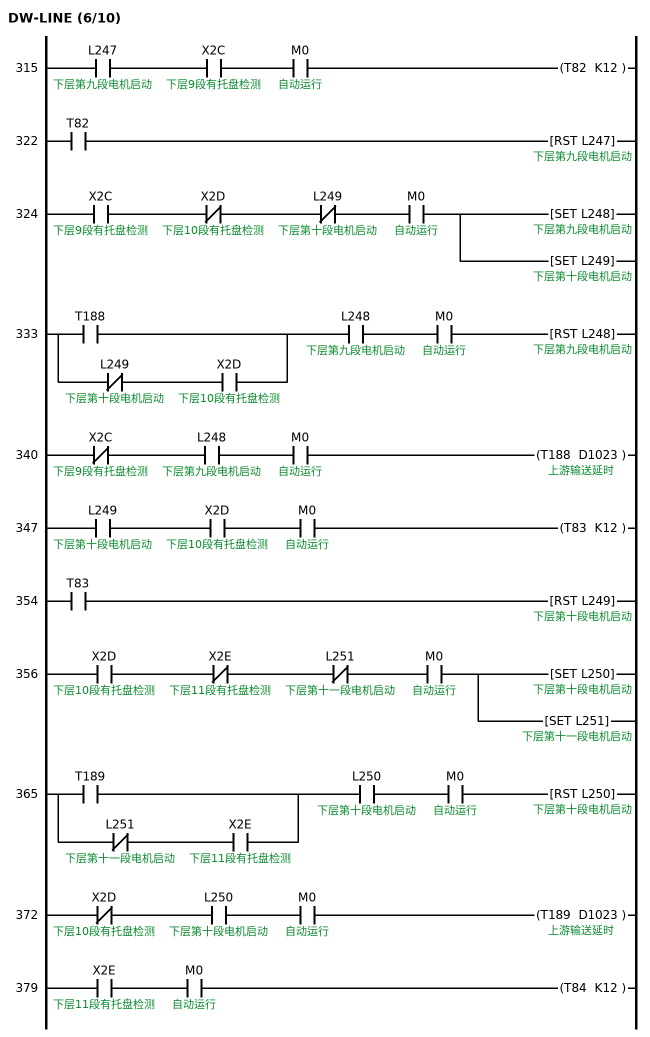
[picture p24: ladder of DW-LINE, rungs at steps 315 to 379]
315   LD      L247  ; 下层第九段电机启动
      AND     X2C  ; 下层9段有托盘检测
      AND     M0  ; 自动运行
      OUT     T82 K12
322   LD      T82
      RST     L247  ; 下层第九段电机启动
324   LD      X2C  ; 下层9段有托盘检测
      ANI     X2D  ; 下层10段有托盘检测
      ANI     L249  ; 下层第十段电机启动
      AND     M0  ; 自动运行
      SET     L248  ; 下层第九段电机启动
        [note] 10
      SET     L249  ; 下层第十段电机启动
333   LD      T188
      LDI     L249  ; 下层第十段电机启动
      AND     X2D  ; 下层10段有托盘检测
      ORB
      AND     L248  ; 下层第九段电机启动
      AND     M0  ; 自动运行
      RST     L248  ; 下层第九段电机启动
340   LDI     X2C  ; 下层9段有托盘检测
      AND     L248  ; 下层第九段电机启动
      AND     M0  ; 自动运行
      OUT     T188 D1023  ; 上游输送延时
347   LD      L249  ; 下层第十段电机启动
      AND     X2D  ; 下层10段有托盘检测
      AND     M0  ; 自动运行
      OUT     T83 K12
354   LD      T83
      RST     L249  ; 下层第十段电机启动
356   LD      X2D  ; 下层10段有托盘检测
      ANI     X2E  ; 下层11段有托盘检测
      ANI     L251  ; 下层第十一段电机启动
      AND     M0  ; 自动运行
      SET     L250  ; 下层第十段电机启动
        [note] 10
      SET     L251  ; 下层第十一段电机启动
365   LD      T189
      LDI     L251  ; 下层第十一段电机启动
      AND     X2E  ; 下层11段有托盘检测
      ORB
      AND     L250  ; 下层第十段电机启动
      AND     M0  ; 自动运行
      RST     L250  ; 下层第十段电机启动
372   LDI     X2D  ; 下层10段有托盘检测
      AND     L250  ; 下层第十段电机启动
      AND     M0  ; 自动运行
      OUT     T189 D1023  ; 上游输送延时
379   LD      X2E  ; 下层11段有托盘检测
      AND     M0  ; 自动运行
      OUT     T84 K12
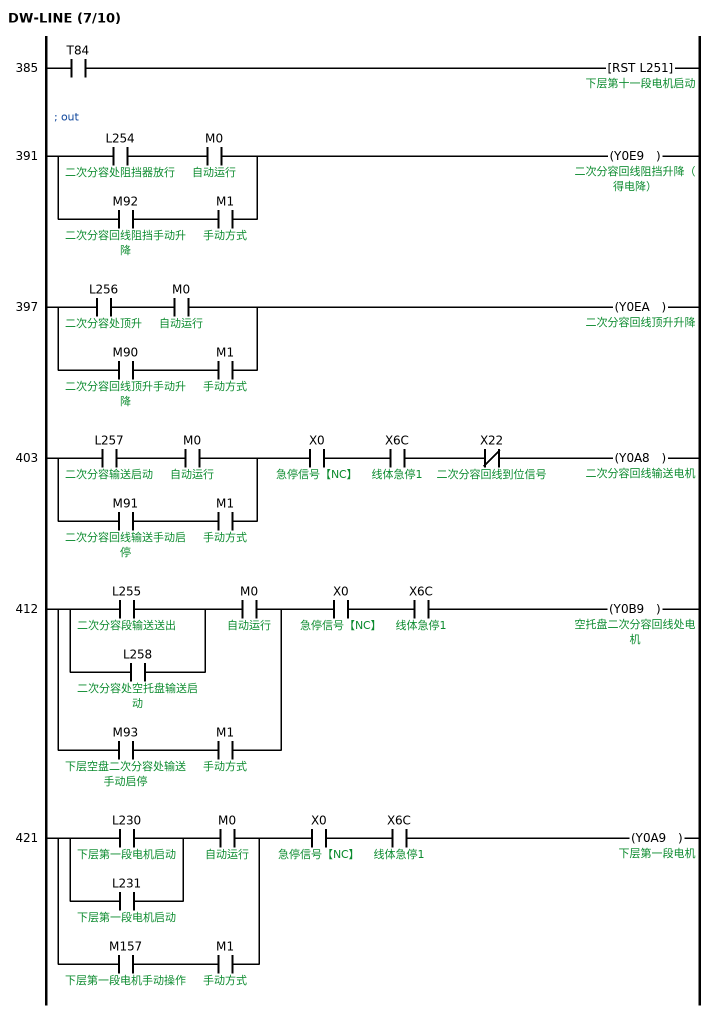
385   LD      T84
      RST     L251  ; 下层第十一段电机启动
; out
391   LD      L254  ; 二次分容处阻挡器放行
      AND     M0  ; 自动运行
      LD      M92  ; 二次分容回线阻挡手动升降
      AND     M1  ; 手动方式
      ORB
      OUT     Y0E9  ; 二次分容回线阻挡升降（得电降）
397   LD      L256  ; 二次分容处顶升
      AND     M0  ; 自动运行
      LD      M90  ; 二次分容回线顶升手动升降
      AND     M1  ; 手动方式
      ORB
      OUT     Y0EA  ; 二次分容回线顶升升降
403   LD      L257  ; 二次分容输送启动
      AND     M0  ; 自动运行
      LD      M91  ; 二次分容回线输送手动启停
      AND     M1  ; 手动方式
      ORB
      AND     X0  ; 急停信号【NC】
      AND     X6C  ; 线体急停1
      ANI     X22  ; 二次分容回线到位信号
      OUT     Y0A8  ; 二次分容回线输送电机
412   LD      L255  ; 二次分容段输送送出
      OR      L258  ; 二次分容处空托盘输送启动
      AND     M0  ; 自动运行
      LD      M93  ; 下层空盘二次分容处输送手动启停
      AND     M1  ; 手动方式
      ORB
      AND     X0  ; 急停信号【NC】
      AND     X6C  ; 线体急停1
      OUT     Y0B9  ; 空托盘二次分容回线处电机
421   LD      L230  ; 下层第一段电机启动
      OR      L231  ; 下层第一段电机启动
      AND     M0  ; 自动运行
      LD      M157  ; 下层第一段电机手动操作
      AND     M1  ; 手动方式
      ORB
      AND     X0  ; 急停信号【NC】
      AND     X6C  ; 线体急停1
      OUT     Y0A9  ; 下层第一段电机
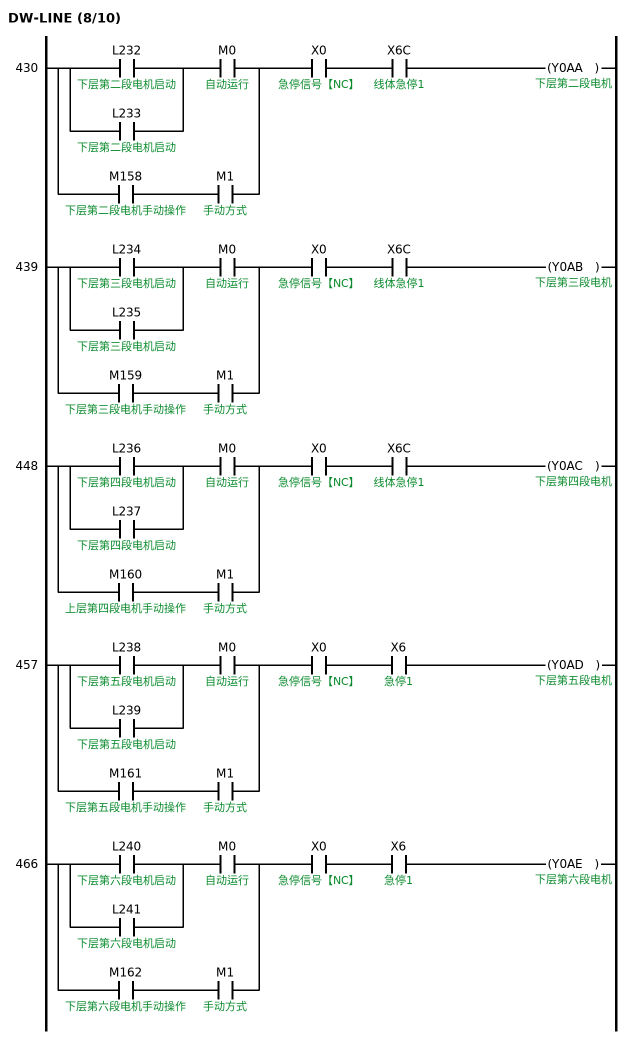
430   LD      L232  ; 下层第二段电机启动
      OR      L233  ; 下层第二段电机启动
      AND     M0  ; 自动运行
      LD      M158  ; 下层第二段电机手动操作
      AND     M1  ; 手动方式
      ORB
      AND     X0  ; 急停信号【NC】
      AND     X6C  ; 线体急停1
      OUT     Y0AA  ; 下层第二段电机
439   LD      L234  ; 下层第三段电机启动
      OR      L235  ; 下层第三段电机启动
      AND     M0  ; 自动运行
      LD      M159  ; 下层第三段电机手动操作
      AND     M1  ; 手动方式
      ORB
      AND     X0  ; 急停信号【NC】
      AND     X6C  ; 线体急停1
      OUT     Y0AB  ; 下层第三段电机
448   LD      L236  ; 下层第四段电机启动
      OR      L237  ; 下层第四段电机启动
      AND     M0  ; 自动运行
      LD      M160  ; 上层第四段电机手动操作
      AND     M1  ; 手动方式
      ORB
      AND     X0  ; 急停信号【NC】
      AND     X6C  ; 线体急停1
      OUT     Y0AC  ; 下层第四段电机
457   LD      L238  ; 下层第五段电机启动
      OR      L239  ; 下层第五段电机启动
      AND     M0  ; 自动运行
      LD      M161  ; 下层第五段电机手动操作
      AND     M1  ; 手动方式
      ORB
      AND     X0  ; 急停信号【NC】
      AND     X6  ; 急停1
      OUT     Y0AD  ; 下层第五段电机
466   LD      L240  ; 下层第六段电机启动
      OR      L241  ; 下层第六段电机启动
      AND     M0  ; 自动运行
      LD      M162  ; 下层第六段电机手动操作
      AND     M1  ; 手动方式
      ORB
      AND     X0  ; 急停信号【NC】
      AND     X6  ; 急停1
      OUT     Y0AE  ; 下层第六段电机
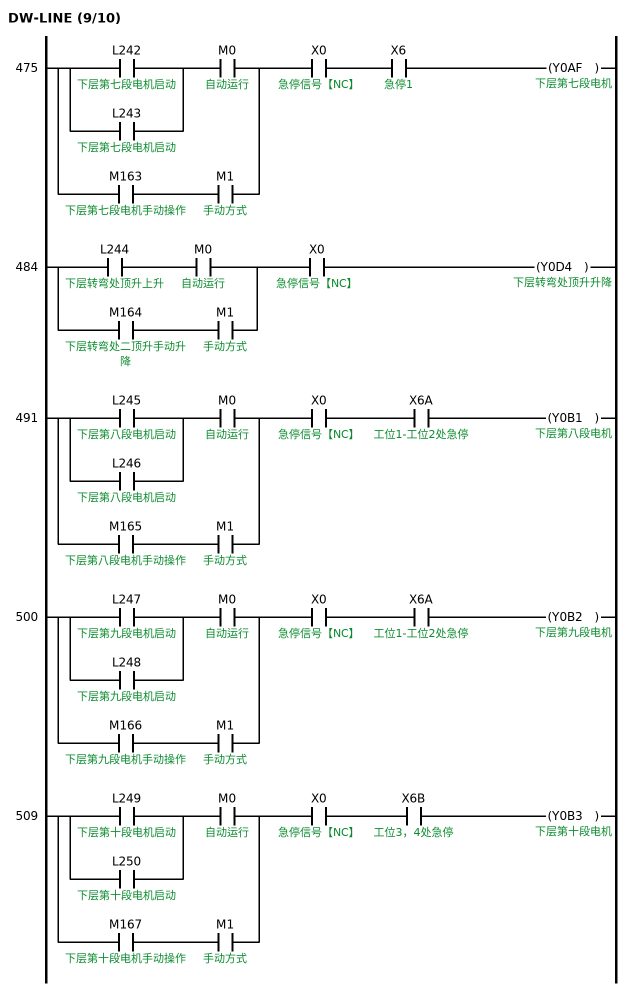
475   LD      L242  ; 下层第七段电机启动
      OR      L243  ; 下层第七段电机启动
      AND     M0  ; 自动运行
      LD      M163  ; 下层第七段电机手动操作
      AND     M1  ; 手动方式
      ORB
      AND     X0  ; 急停信号【NC】
      AND     X6  ; 急停1
      OUT     Y0AF  ; 下层第七段电机
484   LD      L244  ; 下层转弯处顶升上升
      AND     M0  ; 自动运行
      LD      M164  ; 下层转弯处二顶升手动升降
      AND     M1  ; 手动方式
      ORB
      AND     X0  ; 急停信号【NC】
      OUT     Y0D4  ; 下层转弯处顶升升降
491   LD      L245  ; 下层第八段电机启动
      OR      L246  ; 下层第八段电机启动
      AND     M0  ; 自动运行
      LD      M165  ; 下层第八段电机手动操作
      AND     M1  ; 手动方式
      ORB
      AND     X0  ; 急停信号【NC】
      AND     X6A  ; 工位1-工位2处急停
      OUT     Y0B1  ; 下层第八段电机
500   LD      L247  ; 下层第九段电机启动
      OR      L248  ; 下层第九段电机启动
      AND     M0  ; 自动运行
      LD      M166  ; 下层第九段电机手动操作
      AND     M1  ; 手动方式
      ORB
      AND     X0  ; 急停信号【NC】
      AND     X6A  ; 工位1-工位2处急停
      OUT     Y0B2  ; 下层第九段电机
509   LD      L249  ; 下层第十段电机启动
      OR      L250  ; 下层第十段电机启动
      AND     M0  ; 自动运行
      LD      M167  ; 下层第十段电机手动操作
      AND     M1  ; 手动方式
      ORB
      AND     X0  ; 急停信号【NC】
      AND     X6B  ; 工位3，4处急停
      OUT     Y0B3  ; 下层第十段电机
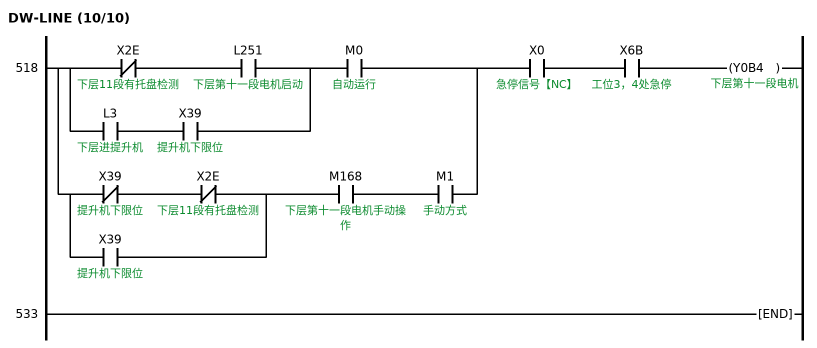
518   LDI     X2E  ; 下层11段有托盘检测
      AND     L251  ; 下层第十一段电机启动
      LD      L3  ; 下层进提升机
      AND     X39  ; 提升机下限位
      ORB
      AND     M0  ; 自动运行
      LDI     X39  ; 提升机下限位
      ANI     X2E  ; 下层11段有托盘检测
      OR      X39  ; 提升机下限位
      AND     M168  ; 下层第十一段电机手动操作
      AND     M1  ; 手动方式
      ORB
      AND     X0  ; 急停信号【NC】
      AND     X6B  ; 工位3，4处急停
      OUT     Y0B4  ; 下层第十一段电机
533   END
END_PROGRAM

PROGRAM ELEVATR
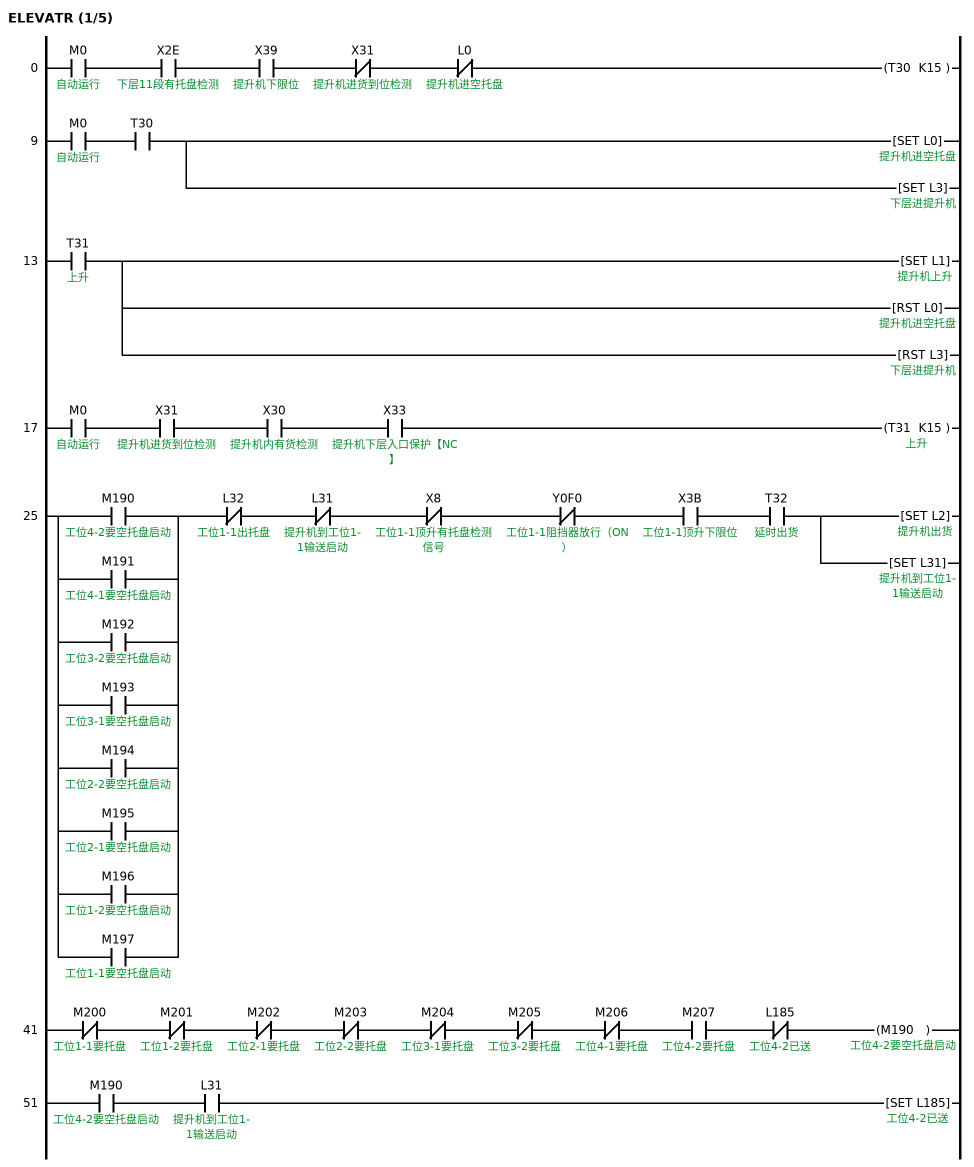
0     LD      M0  ; 自动运行
      AND     X2E  ; 下层11段有托盘检测
      AND     X39  ; 提升机下限位
      ANI     X31  ; 提升机进货到位检测
      ANI     L0  ; 提升机进空托盘
      OUT     T30 K15
9     LD      M0  ; 自动运行
      AND     T30
      SET     L0  ; 提升机进空托盘
      SET     L3  ; 下层进提升机
13    LD      T31  ; 上升
      SET     L1  ; 提升机上升
      RST     L0  ; 提升机进空托盘
      RST     L3  ; 下层进提升机
17    LD      M0  ; 自动运行
      AND     X31  ; 提升机进货到位检测
      AND     X30  ; 提升机内有货检测
      AND     X33  ; 提升机下层入口保护【NC】
      OUT     T31 K15  ; 上升
25    LD      M190  ; 工位4-2要空托盘启动
      OR      M191  ; 工位4-1要空托盘启动
      OR      M192  ; 工位3-2要空托盘启动
      OR      M193  ; 工位3-1要空托盘启动
      OR      M194  ; 工位2-2要空托盘启动
      OR      M195  ; 工位2-1要空托盘启动
      OR      M196  ; 工位1-2要空托盘启动
      OR      M197  ; 工位1-1要空托盘启动
      ANI     L32  ; 工位1-1出托盘
      ANI     L31  ; 提升机到工位1-1输送启动
      ANI     X8  ; 工位1-1顶升有托盘检测信号
      ANI     Y0F0  ; 工位1-1阻挡器放行（ON）
      AND     X3B  ; 工位1-1顶升下限位
      AND     T32  ; 延时出货
      SET     L2  ; 提升机出货
      SET     L31  ; 提升机到工位1-1输送启动
41    LDI     M200  ; 工位1-1要托盘
      ANI     M201  ; 工位1-2要托盘
      ANI     M202  ; 工位2-1要托盘
      ANI     M203  ; 工位2-2要托盘
      ANI     M204  ; 工位3-1要托盘
      ANI     M205  ; 工位3-2要托盘
      ANI     M206  ; 工位4-1要托盘
      AND     M207  ; 工位4-2要托盘
      ANI     L185  ; 工位4-2已送
      OUT     M190  ; 工位4-2要空托盘启动
51    LD      M190  ; 工位4-2要空托盘启动
      AND     L31  ; 提升机到工位1-1输送启动
      SET     L185  ; 工位4-2已送
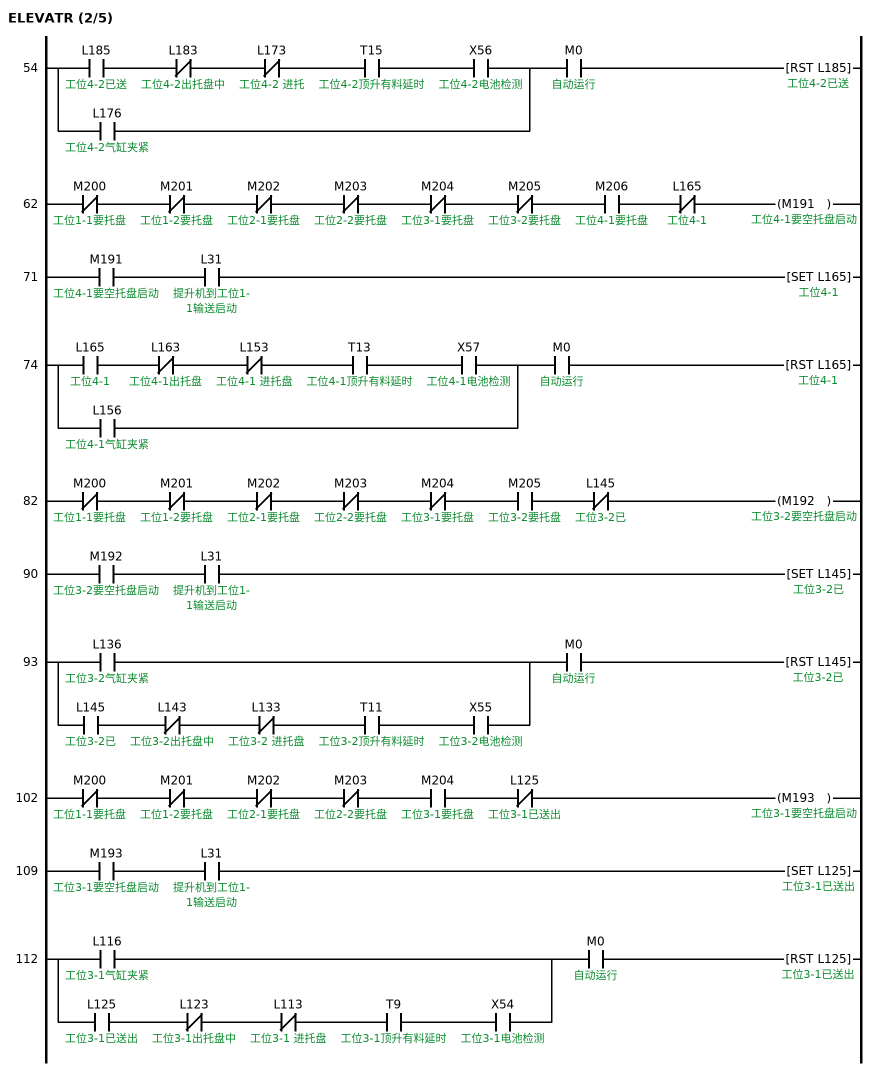
54    LD      L185  ; 工位4-2已送
      ANI     L183  ; 工位4-2出托盘中
      ANI     L173  ; 工位4-2 进托
      AND     T15  ; 工位4-2顶升有料延时
      AND     X56  ; 工位4-2电池检测
      OR      L176  ; 工位4-2气缸夹紧
      AND     M0  ; 自动运行
      RST     L185  ; 工位4-2已送
62    LDI     M200  ; 工位1-1要托盘
      ANI     M201  ; 工位1-2要托盘
      ANI     M202  ; 工位2-1要托盘
      ANI     M203  ; 工位2-2要托盘
      ANI     M204  ; 工位3-1要托盘
      ANI     M205  ; 工位3-2要托盘
      AND     M206  ; 工位4-1要托盘
      ANI     L165  ; 工位4-1
      OUT     M191  ; 工位4-1要空托盘启动
71    LD      M191  ; 工位4-1要空托盘启动
      AND     L31  ; 提升机到工位1-1输送启动
      SET     L165  ; 工位4-1
74    LD      L165  ; 工位4-1
      ANI     L163  ; 工位4-1出托盘
      ANI     L153  ; 工位4-1 进托盘
      AND     T13  ; 工位4-1顶升有料延时
      AND     X57  ; 工位4-1电池检测
      OR      L156  ; 工位4-1气缸夹紧
      AND     M0  ; 自动运行
      RST     L165  ; 工位4-1
82    LDI     M200  ; 工位1-1要托盘
      ANI     M201  ; 工位1-2要托盘
      ANI     M202  ; 工位2-1要托盘
      ANI     M203  ; 工位2-2要托盘
      ANI     M204  ; 工位3-1要托盘
      AND     M205  ; 工位3-2要托盘
      ANI     L145  ; 工位3-2已
      OUT     M192  ; 工位3-2要空托盘启动
90    LD      M192  ; 工位3-2要空托盘启动
      AND     L31  ; 提升机到工位1-1输送启动
      SET     L145  ; 工位3-2已
93    LD      L136  ; 工位3-2气缸夹紧
      LD      L145  ; 工位3-2已
      ANI     L143  ; 工位3-2出托盘中
      ANI     L133  ; 工位3-2 进托盘
      AND     T11  ; 工位3-2顶升有料延时
      AND     X55  ; 工位3-2电池检测
      ORB
      AND     M0  ; 自动运行
      RST     L145  ; 工位3-2已
102   LDI     M200  ; 工位1-1要托盘
      ANI     M201  ; 工位1-2要托盘
      ANI     M202  ; 工位2-1要托盘
      ANI     M203  ; 工位2-2要托盘
      AND     M204  ; 工位3-1要托盘
      ANI     L125  ; 工位3-1已送出
      OUT     M193  ; 工位3-1要空托盘启动
109   LD      M193  ; 工位3-1要空托盘启动
      AND     L31  ; 提升机到工位1-1输送启动
      SET     L125  ; 工位3-1已送出
112   LD      L116  ; 工位3-1气缸夹紧
      LD      L125  ; 工位3-1已送出
      ANI     L123  ; 工位3-1出托盘中
      ANI     L113  ; 工位3-1 进托盘
      AND     T9  ; 工位3-1顶升有料延时
      AND     X54  ; 工位3-1电池检测
      ORB
      AND     M0  ; 自动运行
      RST     L125  ; 工位3-1已送出
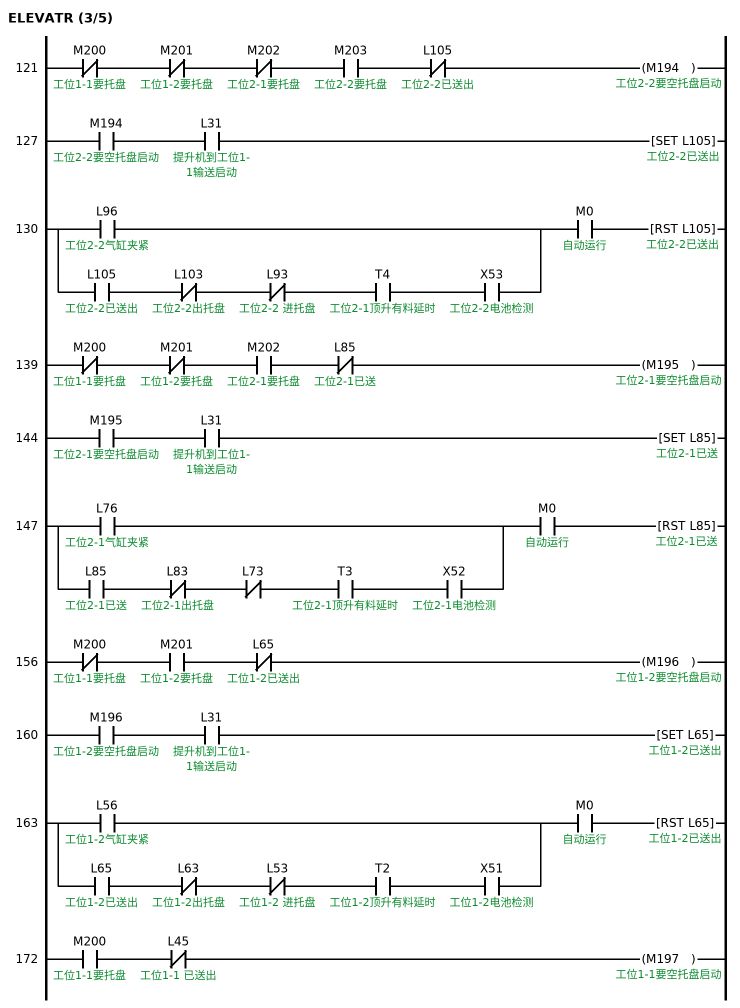
121   LDI     M200  ; 工位1-1要托盘
      ANI     M201  ; 工位1-2要托盘
      ANI     M202  ; 工位2-1要托盘
      AND     M203  ; 工位2-2要托盘
      ANI     L105  ; 工位2-2已送出
      OUT     M194  ; 工位2-2要空托盘启动
127   LD      M194  ; 工位2-2要空托盘启动
      AND     L31  ; 提升机到工位1-1输送启动
      SET     L105  ; 工位2-2已送出
130   LD      L96  ; 工位2-2气缸夹紧
      LD      L105  ; 工位2-2已送出
      ANI     L103  ; 工位2-2出托盘
      ANI     L93  ; 工位2-2 进托盘
      AND     T4  ; 工位2-1顶升有料延时
      AND     X53  ; 工位2-2电池检测
      ORB
      AND     M0  ; 自动运行
      RST     L105  ; 工位2-2已送出
139   LDI     M200  ; 工位1-1要托盘
      ANI     M201  ; 工位1-2要托盘
      AND     M202  ; 工位2-1要托盘
      ANI     L85  ; 工位2-1已送
      OUT     M195  ; 工位2-1要空托盘启动
144   LD      M195  ; 工位2-1要空托盘启动
      AND     L31  ; 提升机到工位1-1输送启动
      SET     L85  ; 工位2-1已送
147   LD      L76  ; 工位2-1气缸夹紧
      LD      L85  ; 工位2-1已送
      ANI     L83  ; 工位2-1出托盘
      ANI     L73
      AND     T3  ; 工位2-1顶升有料延时
      AND     X52  ; 工位2-1电池检测
      ORB
      AND     M0  ; 自动运行
      RST     L85  ; 工位2-1已送
156   LDI     M200  ; 工位1-1要托盘
      AND     M201  ; 工位1-2要托盘
      ANI     L65  ; 工位1-2已送出
      OUT     M196  ; 工位1-2要空托盘启动
160   LD      M196  ; 工位1-2要空托盘启动
      AND     L31  ; 提升机到工位1-1输送启动
      SET     L65  ; 工位1-2已送出
163   LD      L56  ; 工位1-2气缸夹紧
      LD      L65  ; 工位1-2已送出
      ANI     L63  ; 工位1-2出托盘
      ANI     L53  ; 工位1-2 进托盘
      AND     T2  ; 工位1-2顶升有料延时
      AND     X51  ; 工位1-2电池检测
      ORB
      AND     M0  ; 自动运行
      RST     L65  ; 工位1-2已送出
172   LD      M200  ; 工位1-1要托盘
      ANI     L45  ; 工位1-1 已送出
      OUT     M197  ; 工位1-1要空托盘启动
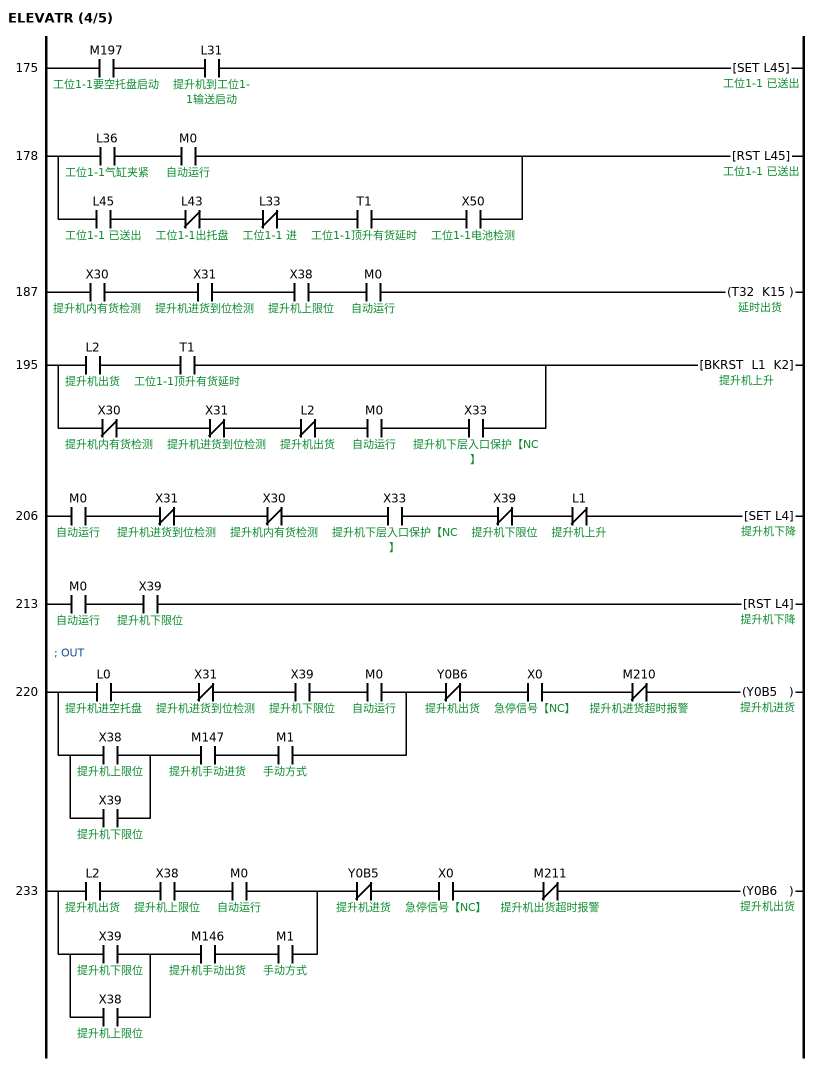
175   LD      M197  ; 工位1-1要空托盘启动
      AND     L31  ; 提升机到工位1-1输送启动
      SET     L45  ; 工位1-1 已送出
178   LD      L36  ; 工位1-1气缸夹紧
      AND     M0  ; 自动运行
      LD      L45  ; 工位1-1 已送出
      ANI     L43  ; 工位1-1出托盘
      ANI     L33  ; 工位1-1 进
      AND     T1  ; 工位1-1顶升有货延时
      AND     X50  ; 工位1-1电池检测
      ORB
      RST     L45  ; 工位1-1 已送出
187   LD      X30  ; 提升机内有货检测
      AND     X31  ; 提升机进货到位检测
      AND     X38  ; 提升机上限位
      AND     M0  ; 自动运行
      OUT     T32 K15  ; 延时出货
195   LD      L2  ; 提升机出货
      AND     T1  ; 工位1-1顶升有货延时
      LDI     X30  ; 提升机内有货检测
      ANI     X31  ; 提升机进货到位检测
      ANI     L2  ; 提升机出货
      AND     M0  ; 自动运行
      AND     X33  ; 提升机下层入口保护【NC】
      ORB
      BKRST   L1 K2
206   LD      M0  ; 自动运行
      ANI     X31  ; 提升机进货到位检测
      ANI     X30  ; 提升机内有货检测
      AND     X33  ; 提升机下层入口保护【NC】
      ANI     X39  ; 提升机下限位
      ANI     L1  ; 提升机上升
      SET     L4  ; 提升机下降
213   LD      M0  ; 自动运行
      AND     X39  ; 提升机下限位
      RST     L4  ; 提升机下降
; OUT
220   LD      L0  ; 提升机进空托盘
      ANI     X31  ; 提升机进货到位检测
      AND     X39  ; 提升机下限位
      AND     M0  ; 自动运行
      LD      X38  ; 提升机上限位
      OR      X39  ; 提升机下限位
      AND     M147  ; 提升机手动进货
      AND     M1  ; 手动方式
      ORB
      ANI     Y0B6  ; 提升机出货
      AND     X0  ; 急停信号【NC】
      ANI     M210  ; 提升机进货超时报警
      OUT     Y0B5  ; 提升机进货
233   LD      L2  ; 提升机出货
      AND     X38  ; 提升机上限位
      AND     M0  ; 自动运行
      LD      X39  ; 提升机下限位
      OR      X38  ; 提升机上限位
      AND     M146  ; 提升机手动出货
      AND     M1  ; 手动方式
      ORB
      ANI     Y0B5  ; 提升机进货
      AND     X0  ; 急停信号【NC】
      ANI     M211  ; 提升机出货超时报警
      OUT     Y0B6  ; 提升机出货
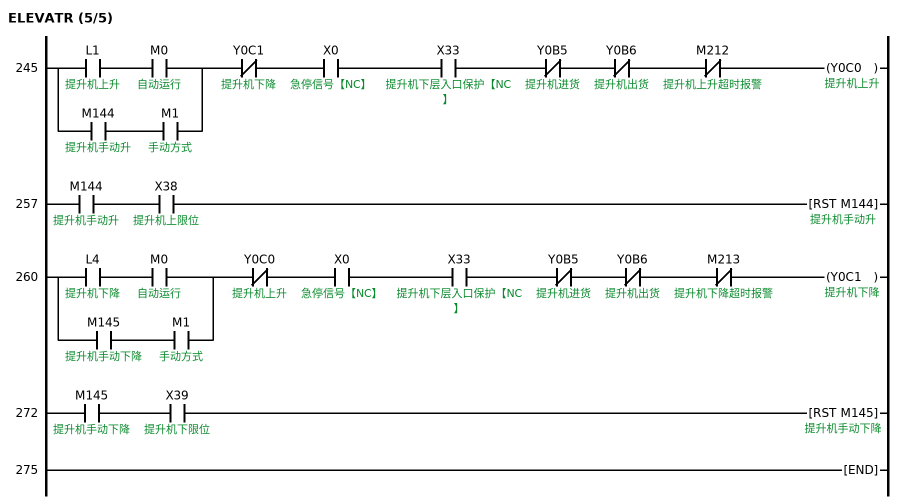
245   LD      L1  ; 提升机上升
      AND     M0  ; 自动运行
      LD      M144  ; 提升机手动升
      AND     M1  ; 手动方式
      ORB
      ANI     Y0C1  ; 提升机下降
      AND     X0  ; 急停信号【NC】
      AND     X33  ; 提升机下层入口保护【NC】
      ANI     Y0B5  ; 提升机进货
      ANI     Y0B6  ; 提升机出货
      ANI     M212  ; 提升机上升超时报警
      OUT     Y0C0  ; 提升机上升
257   LD      M144  ; 提升机手动升
      AND     X38  ; 提升机上限位
      RST     M144  ; 提升机手动升
260   LD      L4  ; 提升机下降
      AND     M0  ; 自动运行
      LD      M145  ; 提升机手动下降
      AND     M1  ; 手动方式
      ORB
      ANI     Y0C0  ; 提升机上升
      AND     X0  ; 急停信号【NC】
      AND     X33  ; 提升机下层入口保护【NC】
      ANI     Y0B5  ; 提升机进货
      ANI     Y0B6  ; 提升机出货
      ANI     M213  ; 提升机下降超时报警
      OUT     Y0C1  ; 提升机下降
272   LD      M145  ; 提升机手动下降
      AND     X39  ; 提升机下限位
      RST     M145  ; 提升机手动下降
275   END
END_PROGRAM

PROGRAM HMI
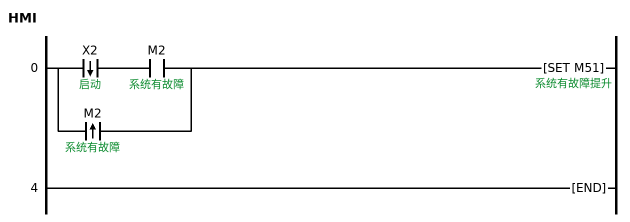
0     LDF     X2  ; 启动
      AND     M2  ; 系统有故障
      ORP     M2  ; 系统有故障
      SET     M51  ; 系统有故障提升
4     END
END_PROGRAM

PROGRAM HMITimer
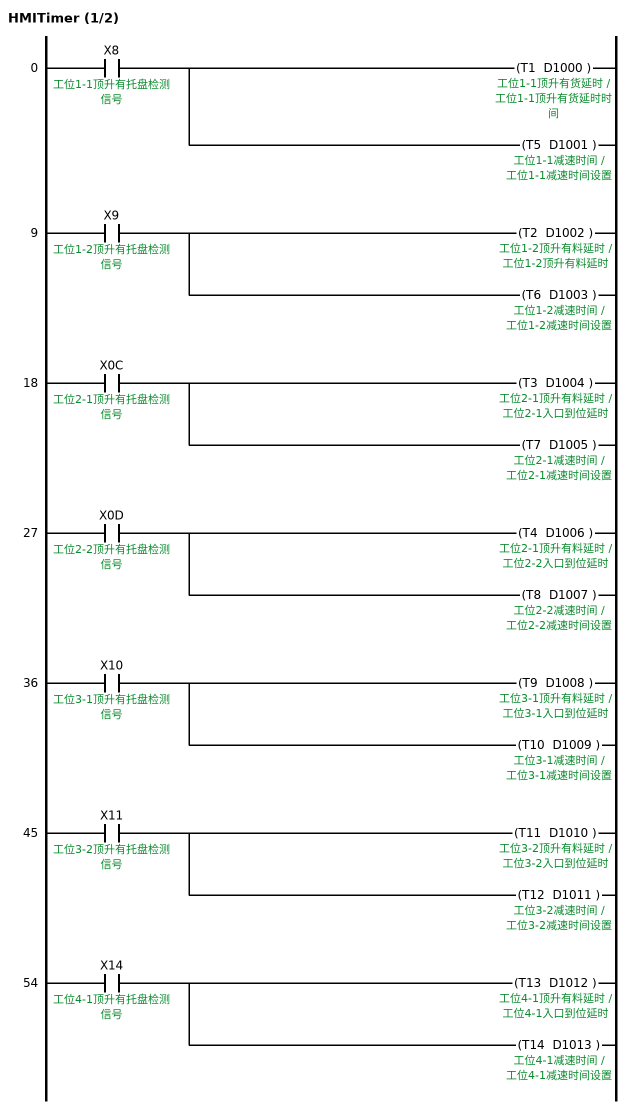
0     LD      X8  ; 工位1-1顶升有托盘检测信号
      OUT     T1 D1000  ; 工位1-1顶升有货延时 / 工位1-1顶升有货延时时间
      OUT     T5 D1001  ; 工位1-1减速时间 / 工位1-1减速时间设置
9     LD      X9  ; 工位1-2顶升有托盘检测信号
      OUT     T2 D1002  ; 工位1-2顶升有料延时 / 工位1-2顶升有料延时
      OUT     T6 D1003  ; 工位1-2减速时间 / 工位1-2减速时间设置
18    LD      X0C  ; 工位2-1顶升有托盘检测信号
      OUT     T3 D1004  ; 工位2-1顶升有料延时 / 工位2-1入口到位延时
      OUT     T7 D1005  ; 工位2-1减速时间 / 工位2-1减速时间设置
27    LD      X0D  ; 工位2-2顶升有托盘检测信号
      OUT     T4 D1006  ; 工位2-1顶升有料延时 / 工位2-2入口到位延时
      OUT     T8 D1007  ; 工位2-2减速时间 / 工位2-2减速时间设置
36    LD      X10  ; 工位3-1顶升有托盘检测信号
      OUT     T9 D1008  ; 工位3-1顶升有料延时 / 工位3-1入口到位延时
      OUT     T10 D1009  ; 工位3-1减速时间 / 工位3-1减速时间设置
45    LD      X11  ; 工位3-2顶升有托盘检测信号
      OUT     T11 D1010  ; 工位3-2顶升有料延时 / 工位3-2入口到位延时
      OUT     T12 D1011  ; 工位3-2减速时间 / 工位3-2减速时间设置
54    LD      X14  ; 工位4-1顶升有托盘检测信号
      OUT     T13 D1012  ; 工位4-1顶升有料延时 / 工位4-1入口到位延时
      OUT     T14 D1013  ; 工位4-1减速时间 / 工位4-1减速时间设置
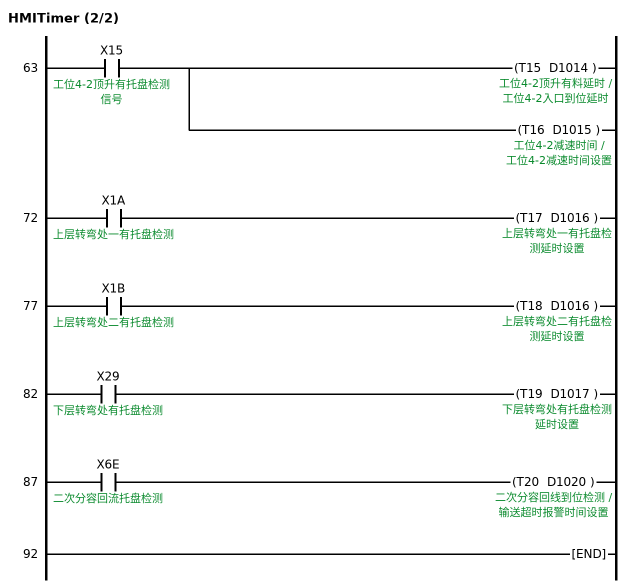
63    LD      X15  ; 工位4-2顶升有托盘检测信号
      OUT     T15 D1014  ; 工位4-2顶升有料延时 / 工位4-2入口到位延时
      OUT     T16 D1015  ; 工位4-2减速时间 / 工位4-2减速时间设置
72    LD      X1A  ; 上层转弯处一有托盘检测
      OUT     T17 D1016  ; 上层转弯处一有托盘检测延时设置
77    LD      X1B  ; 上层转弯处二有托盘检测
      OUT     T18 D1016  ; 上层转弯处二有托盘检测延时设置
82    LD      X29  ; 下层转弯处有托盘检测
      OUT     T19 D1017  ; 下层转弯处有托盘检测延时设置
87    LD      X6E  ; 二次分容回流托盘检测
      OUT     T20 D1020  ; 二次分容回线到位检测 / 输送超时报警时间设置
92    END
END_PROGRAM

PROGRAM INITIALI
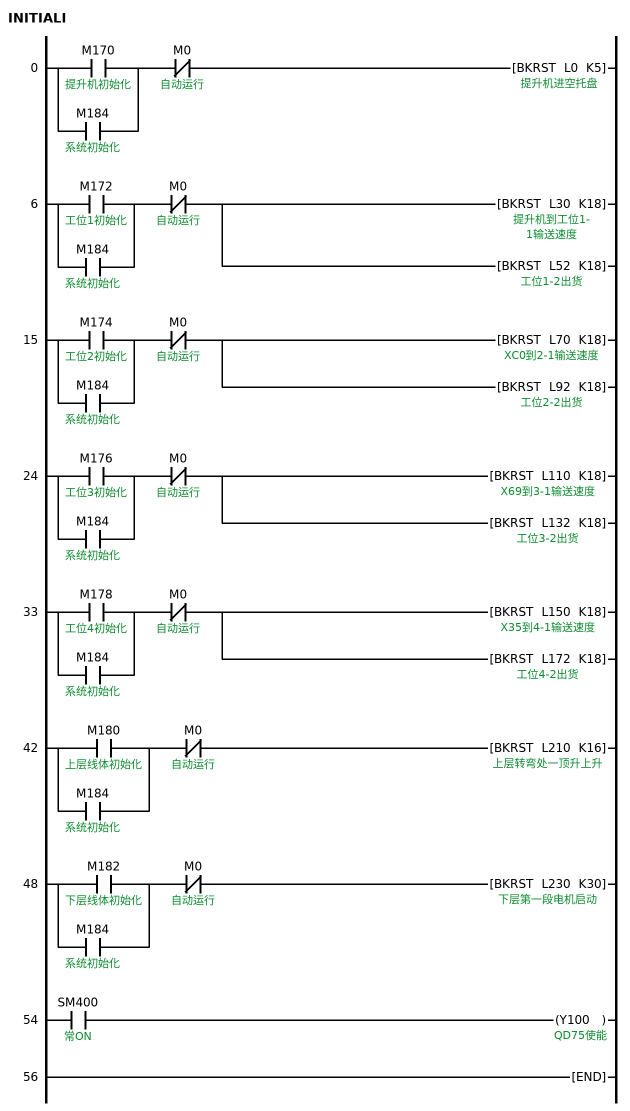
0     LD      M170  ; 提升机初始化
      OR      M184  ; 系统初始化
      ANI     M0  ; 自动运行
      BKRST   L0 K5  ; 提升机进空托盘
6     LD      M172  ; 工位1初始化
      OR      M184  ; 系统初始化
      ANI     M0  ; 自动运行
      BKRST   L30 K18  ; 提升机到工位1-1输送速度
      BKRST   L52 K18  ; 工位1-2出货
15    LD      M174  ; 工位2初始化
      OR      M184  ; 系统初始化
      ANI     M0  ; 自动运行
      BKRST   L70 K18  ; XC0到2-1输送速度
      BKRST   L92 K18  ; 工位2-2出货
24    LD      M176  ; 工位3初始化
      OR      M184  ; 系统初始化
      ANI     M0  ; 自动运行
      BKRST   L110 K18  ; X69到3-1输送速度
      BKRST   L132 K18  ; 工位3-2出货
33    LD      M178  ; 工位4初始化
      OR      M184  ; 系统初始化
      ANI     M0  ; 自动运行
      BKRST   L150 K18  ; X35到4-1输送速度
      BKRST   L172 K18  ; 工位4-2出货
42    LD      M180  ; 上层线体初始化
      OR      M184  ; 系统初始化
      ANI     M0  ; 自动运行
      BKRST   L210 K16  ; 上层转弯处一顶升上升
48    LD      M182  ; 下层线体初始化
      OR      M184  ; 系统初始化
      ANI     M0  ; 自动运行
      BKRST   L230 K30  ; 下层第一段电机启动
54    LD      SM400  ; 常ON
      OUT     Y100  ; QD75使能
56    END
END_PROGRAM

PROGRAM MAIN
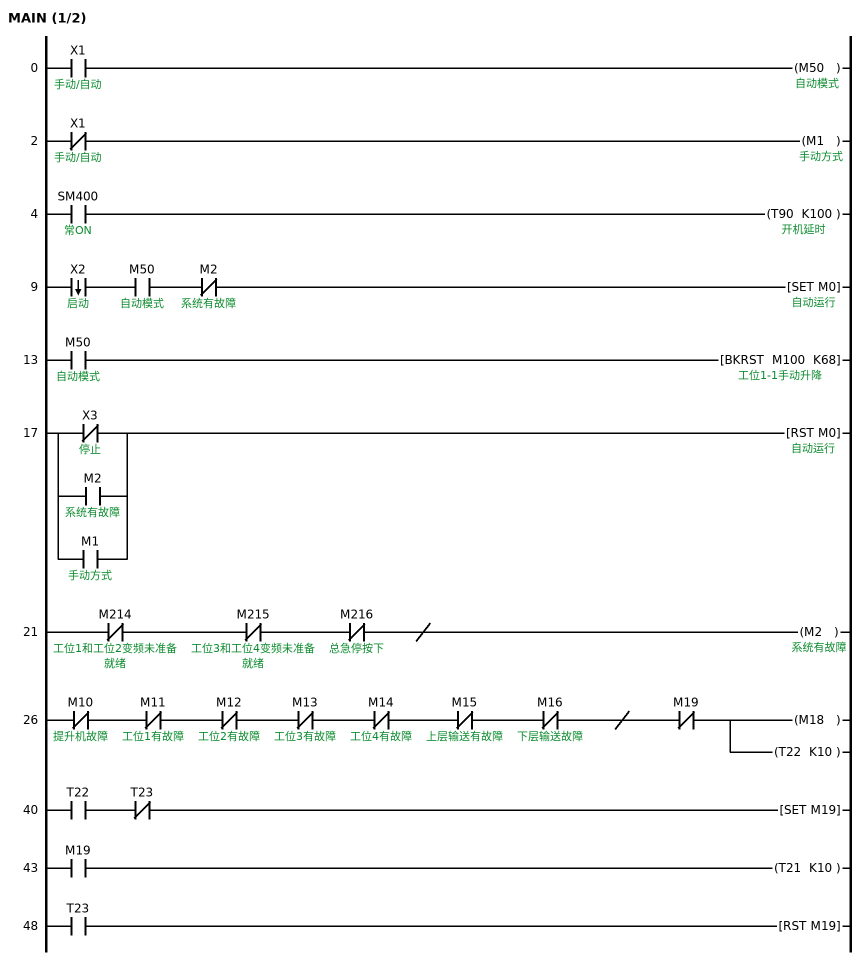
0     LD      X1  ; 手动/自动
      OUT     M50  ; 自动模式
2     LDI     X1  ; 手动/自动
      OUT     M1  ; 手动方式
4     LD      SM400  ; 常ON
      OUT     T90 K100  ; 开机延时
9     LDF     X2  ; 启动
      AND     M50  ; 自动模式
      ANI     M2  ; 系统有故障
      SET     M0  ; 自动运行
13    LD      M50  ; 自动模式
      BKRST   M100 K68  ; 工位1-1手动升降
17    LDI     X3  ; 停止
      OR      M2  ; 系统有故障
      OR      M1  ; 手动方式
      RST     M0  ; 自动运行
21    LDI     M214  ; 工位1和工位2变频未准备就绪
      ANI     M215  ; 工位3和工位4变频未准备就绪
      ANI     M216  ; 总急停按下
      INV
      OUT     M2  ; 系统有故障
26    LDI     M10  ; 提升机故障
      ANI     M11  ; 工位1有故障
      ANI     M12  ; 工位2有故障
      ANI     M13  ; 工位3有故障
      ANI     M14  ; 工位4有故障
      ANI     M15  ; 上层输送有故障
      ANI     M16  ; 下层输送故障
      INV
      ANI     M19
      OUT     M18
      OUT     T22 K10
40    LD      T22
      ANI     T23
      SET     M19
43    LD      M19
      OUT     T21 K10
48    LD      T23
      RST     M19
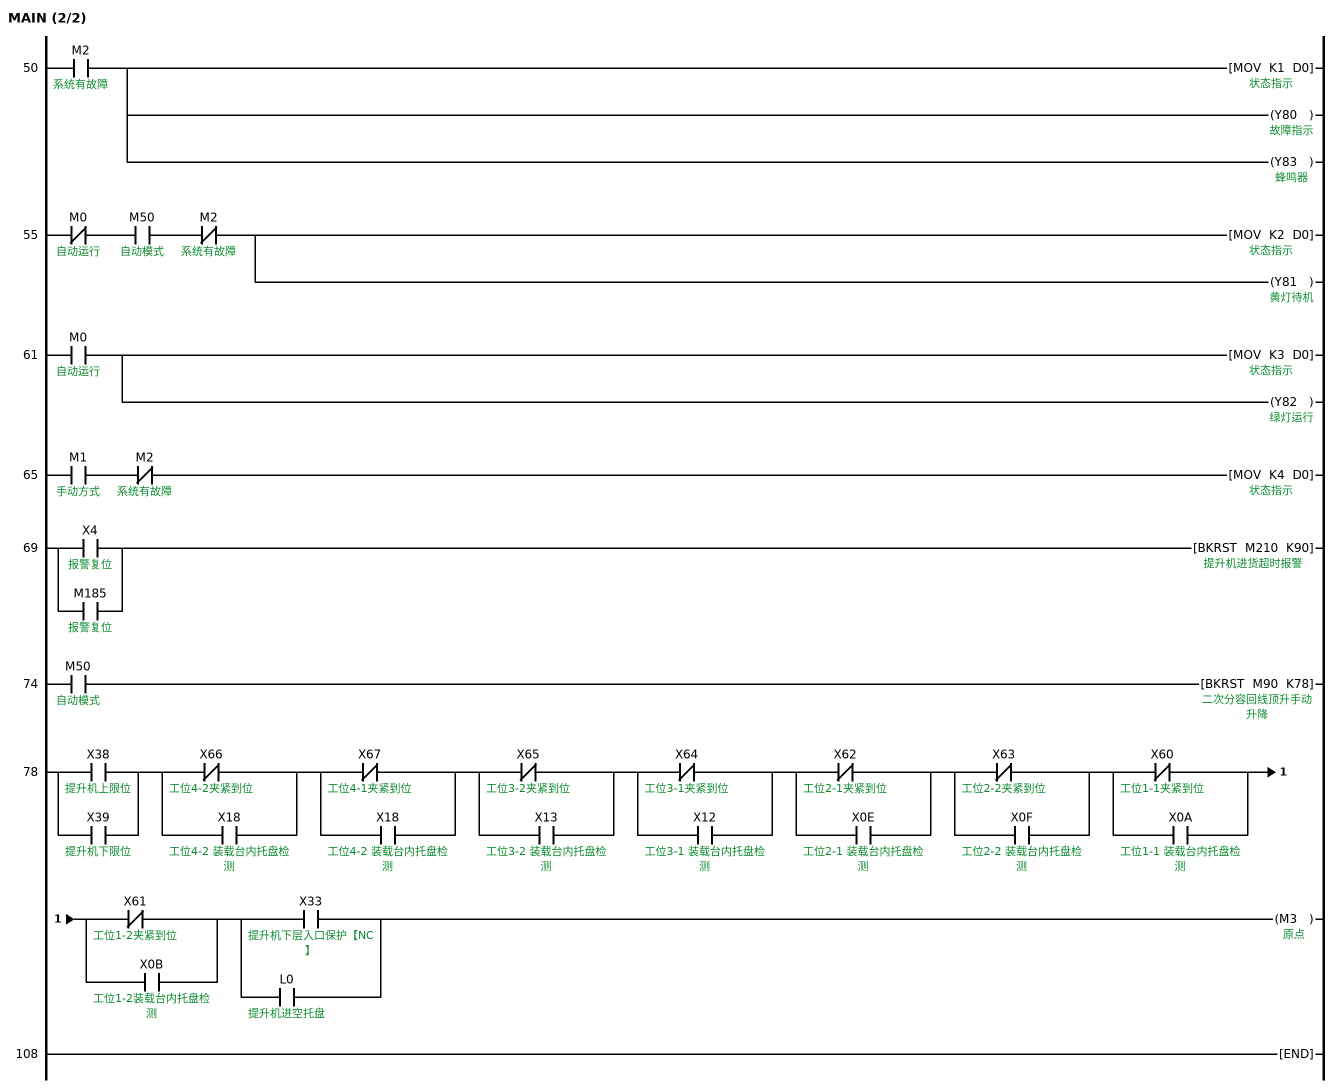
50    LD      M2  ; 系统有故障
      MOV     K1 D0  ; 状态指示
      OUT     Y80  ; 故障指示
      OUT     Y83  ; 蜂鸣器
55    LDI     M0  ; 自动运行
      AND     M50  ; 自动模式
      ANI     M2  ; 系统有故障
      MOV     K2 D0
      OUT     Y81  ; 黄灯待机
61    LD      M0  ; 自动运行
      MOV     K3 D0
      OUT     Y82  ; 绿灯运行
65    LD      M1  ; 手动方式
      ANI     M2  ; 系统有故障
      MOV     K4 D0
69    LD      X4  ; 报警复位
      OR      M185  ; 报警复位
      BKRST   M210 K90  ; 提升机进货超时报警
74    LD      M50  ; 自动模式
      BKRST   M90 K78  ; 二次分容回线顶升手动升降
78    LD      X38  ; 提升机上限位
      OR      X39  ; 提升机下限位
      LDI     X66  ; 工位4-2夹紧到位
      OR      X18  ; 工位4-2 装载台内托盘检测
      ANB
      LDI     X67  ; 工位4-1夹紧到位
      OR      X18  ; 工位4-2 装载台内托盘检测
      ANB
      LDI     X65  ; 工位3-2夹紧到位
      OR      X13  ; 工位3-2 装载台内托盘检测
      ANB
      LDI     X64  ; 工位3-1夹紧到位
      OR      X12  ; 工位3-1 装载台内托盘检测
      ANB
      LDI     X62  ; 工位2-1夹紧到位
      OR      X0E  ; 工位2-1 装载台内托盘检测
      ANB
      LDI     X63  ; 工位2-2夹紧到位
      OR      X0F  ; 工位2-2 装载台内托盘检测
      ANB
      LDI     X60  ; 工位1-1夹紧到位
      OR      X0A  ; 工位1-1 装载台内托盘检测
      ANB
      LDI     X61  ; 工位1-2夹紧到位
      OR      X0B  ; 工位1-2装载台内托盘检测
      ANB
      LD      X33  ; 提升机下层入口保护【NC】
      OR      L0  ; 提升机进空托盘
      ANB
      OUT     M3  ; 原点
108   END
END_PROGRAM

PROGRAM PRODUCT
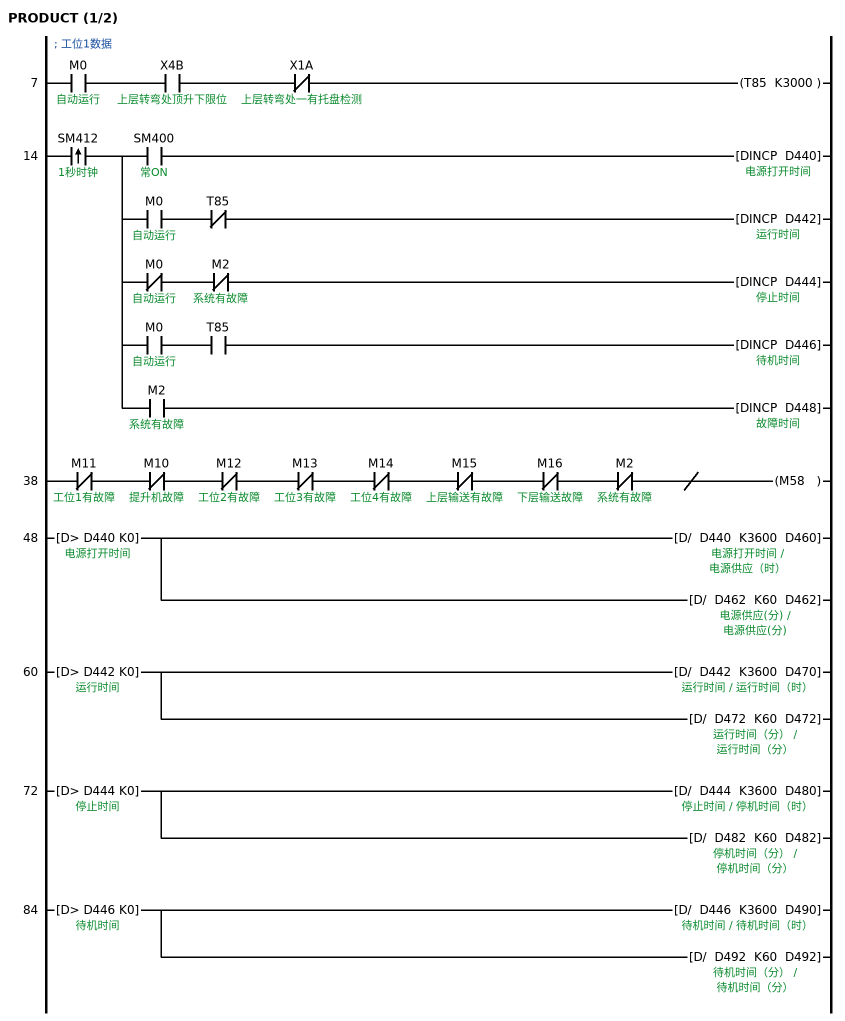
; 工位1数据
7     LD      M0  ; 自动运行
      AND     X4B  ; 上层转弯处顶升下限位
      ANI     X1A  ; 上层转弯处一有托盘检测
      OUT     T85 K3000
14    LDP     SM412  ; 1秒时钟
      MPS
      AND     SM400  ; 常ON
      DINCP   D440  ; 电源打开时间
      MRD
      AND     M0  ; 自动运行
      ANI     T85
      DINCP   D442  ; 运行时间
      MRD
      ANI     M0  ; 自动运行
      ANI     M2  ; 系统有故障
      DINCP   D444  ; 停止时间
      MRD
      AND     M0  ; 自动运行
      AND     T85
      DINCP   D446  ; 待机时间
      MPP
      AND     M2  ; 系统有故障
      DINCP   D448  ; 故障时间
38    LDI     M11  ; 工位1有故障
      ANI     M10  ; 提升机故障
      ANI     M12  ; 工位2有故障
      ANI     M13  ; 工位3有故障
      ANI     M14  ; 工位4有故障
      ANI     M15  ; 上层输送有故障
      ANI     M16  ; 下层输送故障
      ANI     M2  ; 系统有故障
      INV
      OUT     M58
48    LDD>    D440 K0  ; 电源打开时间
      D/      D440 K3600 D460  ; 电源供应（时）
      D/      D462 K60 D462  ; 电源供应(分)
60    LDD>    D442 K0  ; 运行时间
      D/      D442 K3600 D470  ; 运行时间（时）
      D/      D472 K60 D472  ; 运行时间（分）
72    LDD>    D444 K0  ; 停止时间
      D/      D444 K3600 D480  ; 停机时间（时）
      D/      D482 K60 D482  ; 停机时间（分）
84    LDD>    D446 K0  ; 待机时间
      D/      D446 K3600 D490  ; 待机时间（时）
      D/      D492 K60 D492  ; 待机时间（分）
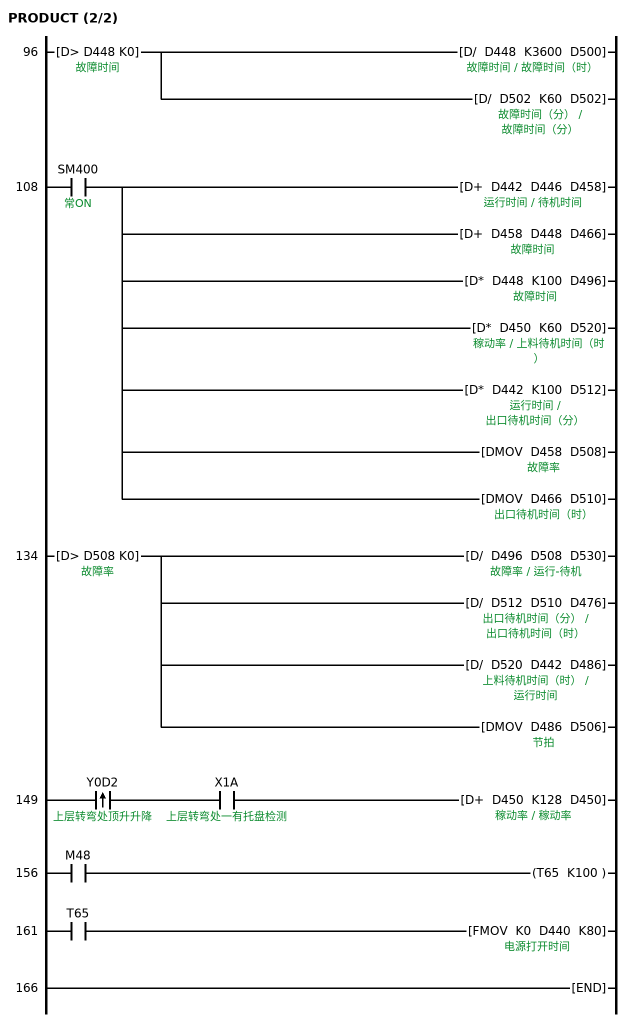
96    LDD>    D448 K0  ; 故障时间
      D/      D448 K3600 D500  ; 故障时间（时）
      D/      D502 K60 D502  ; 故障时间（分）
108   LD      SM400  ; 常ON
      D+      D442 D446 D458
        [note] 秒
      D+      D458 D448 D466
      D*      D448 K100 D496
      D*      D450 K60 D520  ; 稼动率 / 上料待机时间（时）
      D*      D442 K100 D512  ; 出口待机时间（分）
      DMOV    D458 D508  ; 故障率
      DMOV    D466 D510  ; 出口待机时间（时）
134   LDD>    D508 K0  ; 故障率
      D/      D496 D508 D530  ; 运行-待机
      D/      D512 D510 D476
      D/      D520 D442 D486
      DMOV    D486 D506  ; 节拍
149   LDP     Y0D2  ; 上层转弯处顶升升降
      AND     X1A  ; 上层转弯处一有托盘检测
      D+      D450 K128 D450
156   LD      M48
      OUT     T65 K100
161   LD      T65
      FMOV    K0 D440 K80
166   END
END_PROGRAM

PROGRAM ServoScan
VAR
  istep : INT;  (* 扫码步骤 *)
END_VAR
VAR CONSTANT
  ROW : INT := 8;  (* Y轴每个值对应的电池数量 *)
END_VAR
VAR
  ii : INT;
  jj : INT;
  m_xclean : BOOL;  (* 清零 *)
  kk : INT;  (* 错误位 *)
  m_iLampTwinkle : INT;  (* 灯光闪烁次数 *)
END_VAR
(*当前位置读取*)
DMOVP(SM412,g_diQD75CurrentPos1,g_diQD75LastPos1);(*记录1S前的位置，和现在的位置比较，判断是否需要重新启动*)
DMOVP(SM412,g_diQD75CurrentPos2,g_diQD75LastPos2);(*记录1S前的位置，和现在的位置比较，判断是否需要重新启动*)
DMOVP(SM412,U10\G800,g_diQD75CurrentPos1);(*双字不能:=，只能dmov了*)
DMOVP(SM412,U10\G900,g_diQD75CurrentPos2);(*双字不能:=，只能dmov了*)
(*如果Y有输出，但是电机没走，那可能是定位过程中发了新的指令，就用这个来断一下Y就能恢复动作了*)
IF (g_yQD75LocateStart1 AND g_diQD75CurrentPos1=g_diQD75LastPos1 )
	 OR (g_yQD75LocateStart2 AND g_diQD75CurrentPos2=g_diQD75LastPos2 ) THEN
				g_xResetServo:=1;
ELSE
				g_xResetServo:=0;
END_IF;		
(*目标地址读取*)
g_iQD75LastNumber1:=U10\G837;(*上一次目标号*)
g_iQD75DestiNumber1:=U10\G835;(*目标号*)
DMOV(TRUE,U10\G818,g_diQD75DestinationPos1);(*目标地址*)
g_iQD75LastNumber2:=U10\G937;(*上一次目标号*)
g_iQD75DestiNumber2:=U10\G935;(*目标号*)
DMOV(TRUE,U10\G918,g_diQD75DestinationPos2);(*目标地址*)
(*报警信息读取*)
g_iQD75ErrorNumber1:=U10\G806;
g_iQD75ErrorNumber2:=U10\G906;
(*报警复位*)
IF LDP(TRUE,g_xResetServo) THEN
	U10\G1502:=1;(*X轴复位*)(*这俩信号都能自动复位*)
	U10\G1602:=1;(*Y轴复位*)
	U10\G1503:=1;(*X轴重起*)
	U10\G1603:=1;(*Y轴重起*)
	YFE:= X78 OR  X79;(*X78,X79为两个驱动器的报警，这个驱动器只能断电复位，所以YAE控制断电*)
ELSE
	YFE:=0;
	
END_IF;	







(*下面是正式流程*)
(*除了正常运过去那种，有时手动放上去的也要能启动扫码流程，要加个按钮*)
SET( g_xPutInto, g_xServoStart );
 CASE istep OF 
 0:(*初始化，等待启动信号*)
 				U10\G1500:=9001;(*9001表示会回原点*)
 				U10\G1600:=9001;
 				(*g_yQD75LocateStart1:= NOT g_xResetServo AND NOT g_xQD75LocateDone1
 																AND U10\G800<>0;
 				g_yQD75LocateStart2:= NOT g_xResetServo AND NOT g_xQD75LocateDone2
 																AND U10\G900<>0;		*)
 				MOV( g_xServoStart AND U10\G800=0 AND U10\G900=0, 10, istep );(*800是当前位置值*)
 	(*10是在0之后，1之前的一个步骤，扫框码，等待扫码完成。懒得改，就插在这里了*)
 10:(*扫框码，扫码完成再去扫电池码*)
 				(*夹紧气缸夹住*)
 				g_yQD75LocateStart1:=0;
 				g_yQD75LocateStart2:=0;
 				g_xCatchCylinder:=1;
 	 			g_xServoStart:=0;
 				g_xScan:=0; 	
 				D3000:=2;(**扫框码请求**)
 				IF D2000=2 THEN(*扫码成功*)
 							g_iXaxisNumber:=1;
 							g_iYaxisNumber:=1;
 							istep:=1;
 				END_IF;	
 1:(*伺服行走*)
 				(*X轴行走*)	
 				IF NOT g_xQD75LocateDone1 AND g_iXaxisNumber<>0 THEN(*起始地址设定是100，那么g_xQD75LocateDone1就是1轴定位完成信号*)
 							U10\G1500:=g_iXaxisNumber;(*起始地址设定是100，这里就要写U10，起始地址去掉个0。G1500是X轴定位启动的编号*)
 							g_yQD75LocateStart1:=NOT g_xResetServo;(*起始地址设定是100，那么g_yQD75LocateStart1就是1轴定位启动信号*)
 				ELSE
 							U10\G1500:=0;
 							g_yQD75LocateStart1:=0;
 				END_IF;		
 				(*Y轴行走*)	
 				IF NOT g_xQD75LocateDone2 AND g_iYaxisNumber<>0 THEN
 							U10\G1600:=g_iYaxisNumber;
 							g_yQD75LocateStart2:=NOT g_xResetServo;
 				ELSE
 							U10\G1600:=0;
 							g_yQD75LocateStart2:=0;
 				END_IF;	
 				SET( g_xQD75LocateDone1 AND g_xQD75LocateDone2 , g_xScan);
 				SET( g_xQD75LocateDone1 AND g_xQD75LocateDone2 , g_xScan1); 				
 				SET( g_xQD75LocateDone1 AND g_xQD75LocateDone2 AND g_iXaxisNumber<>3, g_xScan2); 				
 				MOV( g_xQD75LocateDone1 AND g_xQD75LocateDone2 , 2, istep );
 2:(*进行扫码*)
 				g_yQD75LocateStart1:=0;
 				g_yQD75LocateStart2:=0;
 				(*扫码结果为8，表示扫码错误，调回step1，重新扫一次*)
 				IF g_iBatteryInformation[0]=8 AND TS67 THEN
 							g_iBatteryInformation[0]:=0;
 							g_xScan:=0;
							FOR ii:=0 TO 10 DO
 													IF g_iScanError[ii]=0 THEN(*把错误字都存起来，完成任务清零*)
 															g_iScanError[ii]:=g_iBatteryPosition;
 															g_iErrorSUM:=ii+1;
 															EXIT;
 													END_IF;
 							END_FOR;		
 							IF g_iBatteryPosition>0 AND g_iBatteryPosition<128 AND TS67 THEN
 										(*数据复位*)
 													FOR jj:=0 TO 16 DO
 															g_iBatteryInformation[jj]:=0;
 													END_FOR;
 										(*这里的框是特殊形状的，有16列，每列对应8排，但是基数列和偶数列又是错开的，所以单独写的位置计算*)
 				 									g_iBatteryPosition:=g_iBatteryPosition+1;
 													g_iXaxisNumber:=(g_iBatteryPosition-1)/ROW+1;
 													g_iYaxisNumber:=2*((g_iBatteryPosition-1)MOD ROW)+1+((g_iXaxisNumber-1) MOD 2);(*后面这个是判断奇偶的，奇数列不加，偶数列加1*)
 													istep:=1;
 							ELSIF g_iBatteryPosition=128 AND TS67 THEN
 													FOR jj:=0 TO 16 DO
 																g_iBatteryInformation[jj]:=0;
 													END_FOR;
 													istep:=3;	
 							END_IF;			

 						(*	END_IF;	*)
 				END_IF;	
 				Z0:=(g_iBatteryPosition-1)*15;(*正常情况，每个电池占用15个字,-1是因为位置参数是从1开始，不是0开始*)
 				IF g_xScan AND g_iBatteryInformation[0]=24 THEN(*扫码成功会有24个字，不成功会有8个字，还可能读错，就会超过24个字，都属于不正常*)
 							D3006Z0:=g_iBatteryInformation[1];
 							D3007Z0:=g_iBatteryInformation[2];(*1-14都是电池码*)
 							D3008Z0:=g_iBatteryInformation[3];
 							D3009Z0:=g_iBatteryInformation[4];
 							D3010Z0:=g_iBatteryInformation[5];
 							D3011Z0:=g_iBatteryInformation[6];
 							D3012Z0:=g_iBatteryInformation[7];
 							D3013Z0:=g_iBatteryInformation[8];
 							D3014Z0:=g_iBatteryInformation[9];
 							D3015Z0:=g_iBatteryInformation[10];
 							D3016Z0:=g_iBatteryInformation[11];
 							D3017Z0:=g_iBatteryInformation[12];
 							D3018Z0:=g_iBatteryInformation[13];
 							D3019Z0:=g_iBatteryInformation[14];
 							D3020Z0:=g_iBatteryInformation[15];
 							IF g_iBatteryPosition>0 AND g_iBatteryPosition<128 AND TS67 THEN
 										g_xScan:=0;
 										(*数据复位*)
 										FOR jj:=0 TO 16 DO
 													g_iBatteryInformation[jj]:=0;
 										END_FOR;
 										(*这里的框是特殊形状的，有16列，每列对应8排，但是基数列和偶数列又是错开的，所以单独写的位置计算*)
 				 						g_iBatteryPosition:=g_iBatteryPosition+1;
 										g_iXaxisNumber:=(g_iBatteryPosition-1)/ROW+1;
 										g_iYaxisNumber:=2*((g_iBatteryPosition-1)MOD ROW)+1+((g_iXaxisNumber-1) MOD 2);(*后面这个是判断奇偶的，奇数列不加，偶数列加1*)
 										istep:=1;
 						ELSIF g_iBatteryPosition=128 AND TS67 THEN
 										FOR jj:=0 TO 16 DO
 													g_iBatteryInformation[jj]:=0;
 										END_FOR;
 										g_xScan:=0;
 										istep:=3;	
 						END_IF;(*位置在1-128之间那个if*)
 				END_IF;(*扫码成功那个if*)		
 3:(*数据上传*)
   				IF g_iScanError[6]=0 THEN
 							D3001:=2;(*装载完成，数据上传*)
 				END_IF;
 				IF D2001=2 THEN(*表示数据收到，可以放行*)
 							istep:=4;
 				END_IF;
 4:(*数据复位，下料，回0步*)
 				D3001:=1;
 				g_xCatchCylinder:=0;
 				g_xScanDone:=1;
 				IF X100 THEN
 							U10\G1500:=1;
 							U10\G1600:=1;
 							g_yQD75LocateStart1:=NOT g_xQD75LocateDone1 AND NOT g_xResetServo;
 							g_yQD75LocateStart2:=NOT g_xQD75LocateDone2 AND NOT g_xResetServo;
 				END_IF;
 20:(*这里加一个专门去不良位的，调试用*)
 				 D2009:=g_iScanError[0]+g_iScanError[1](*这个没有意义，只是为了方便我看没扫上的那些位置*)
 								+g_iScanError[2]+g_iScanError[3]+g_iScanError[ 4]
								+g_iScanError[5] +g_iScanError[6] +g_iScanError[7]
  								+g_iScanError[8]+g_iScanError[9];
 				g_iXaxisNumber:=(kk-1)/ROW+1;
 				g_iYaxisNumber:=2*((kk-1)MOD ROW)+1+((g_iXaxisNumber-1) MOD 2);
 				U10\G1500:=g_iXaxisNumber;
 				U10\G1600:=g_iYaxisNumber; 
 				DMOV(TRUE,10000,U10\G1518);
 				DMOV(TRUE,10000,U10\G1618);
 				g_yQD75LocateStart1:=NOT g_xQD75LocateDone1 AND NOT g_yQD75JogCW1 AND NOT g_yQD75JogCCW1 AND NOT g_xResetServo;
 				g_yQD75LocateStart2:=NOT g_xQD75LocateDone2 AND NOT g_yQD75JogCW2 AND NOT g_yQD75JogCCW2 AND NOT g_xResetServo;
 				g_yQD75JogCW1:=NOT g_yQD75JogCCW1 AND g_xJogXCW;(*1轴JOG正转*)
 				g_yQD75JogCCW1:=NOT g_yQD75JogCW1 AND g_xJogXCCW;(*1轴JOG反转*)
 				g_yQD75JogCW2:=NOT g_yQD75JogCCW2 AND g_xJogYCW;(*2轴JOG正转*)
 				g_yQD75JogCCW2:=NOT g_yQD75JogCW2 AND g_xJogYCCW;(*2轴JOG反转*)
 				
 END_CASE;
(*这个写在case外边，方便复位*) 
IF TS190 AND NOT g_xQD75Busy1 AND NOT g_xQD75Busy2 THEN
	(*T190是下料时，离开开关延时，离开开关这么久就认为物料已远走，可以开始运下一个了*)
 			FOR Z1:=0 TO 1920 DO(*物料送走，数据复位*)
 						D3006Z1:=0;
 		 	END_FOR;
 		  	D3000:=1;(*扫框码请求复位*)
 		  	g_xServoStart:=0;
 			g_xScanDone:=0;
 			g_iBatteryPosition:=1;
 		(*	istep:=0;*)
END_IF;
 OUT_T( g_iBatteryInformation[0]<>0 AND istep=2,TC67 ,k3 );(*扫码成功到接收数据完毕需要时间，所以做个延时*)
 OUT_T( g_iBatteryInformation[0]=0 AND istep=2 ,TC66 ,k100);(*有时候扫码请求发出去数据没接收到，需要重新启动扫码，等10S*)
 IF TS190 OR m_xclean THEN
 	FOR jj:=0 TO 9 DO
 		g_iScanError[jj]:=0;
 	END_FOR;
 	g_iErrorSUM:=0;
 END_IF;		
 YBA:=g_iScanError[6]<>0;(*超过6个就报警*)
END_PROGRAM

PROGRAM STATION1
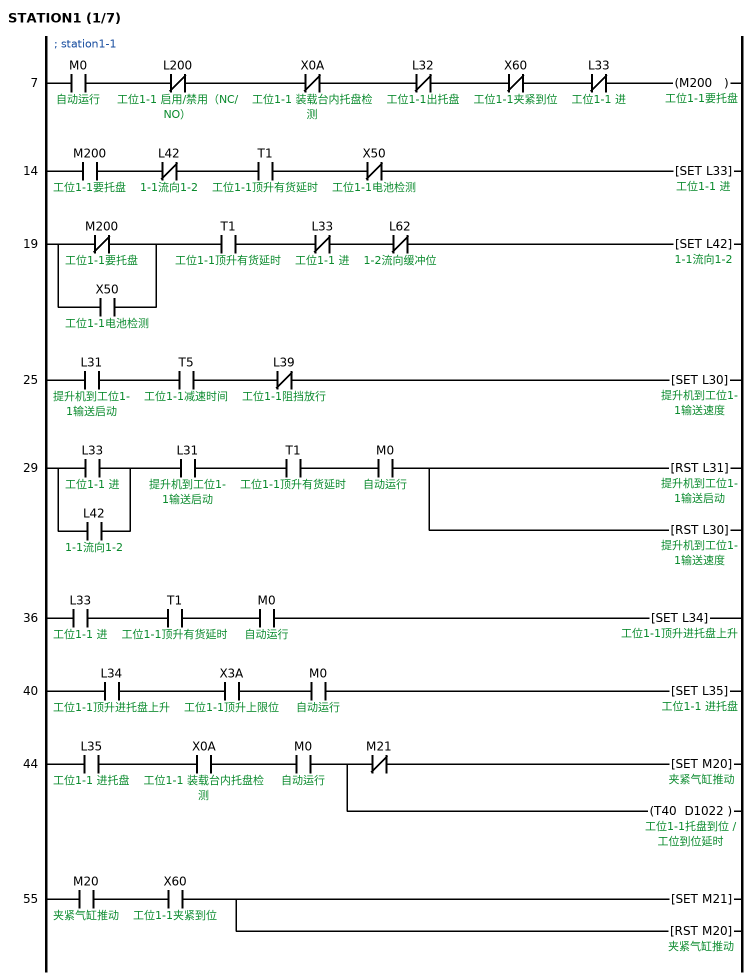
; station1-1
7     LD      M0  ; 自动运行
      ANI     L200  ; 工位1-1 启用/禁用（NC/NO）
      ANI     X0A  ; 工位1-1 装载台内托盘检测
      ANI     L32  ; 工位1-1出托盘
      ANI     X60  ; 工位1-1夹紧到位
      ANI     L33  ; 工位1-1 进
      OUT     M200  ; 工位1-1要托盘
14    LD      M200  ; 工位1-1要托盘
      ANI     L42  ; 1-1流向1-2
      AND     T1  ; 工位1-1顶升有货延时
      ANI     X50  ; 工位1-1电池检测
      SET     L33  ; 工位1-1 进
19    LDI     M200  ; 工位1-1要托盘
      OR      X50  ; 工位1-1电池检测
      AND     T1  ; 工位1-1顶升有货延时
      ANI     L33  ; 工位1-1 进
      ANI     L62  ; 1-2流向缓冲位
      SET     L42  ; 1-1流向1-2
25    LD      L31  ; 提升机到工位1-1输送启动
      AND     T5  ; 工位1-1减速时间
      ANI     L39  ; 工位1-1阻挡放行
      SET     L30  ; 提升机到工位1-1输送速度
29    LD      L33  ; 工位1-1 进
      OR      L42  ; 1-1流向1-2
      AND     L31  ; 提升机到工位1-1输送启动
      AND     T1  ; 工位1-1顶升有货延时
      AND     M0  ; 自动运行
      RST     L31  ; 提升机到工位1-1输送启动
      RST     L30  ; 提升机到工位1-1输送速度
36    LD      L33  ; 工位1-1 进
      AND     T1  ; 工位1-1顶升有货延时
      AND     M0  ; 自动运行
      SET     L34  ; 工位1-1顶升进托盘上升
40    LD      L34  ; 工位1-1顶升进托盘上升
      AND     X3A  ; 工位1-1顶升上限位
      AND     M0  ; 自动运行
      SET     L35  ; 工位1-1 进托盘
44    LD      L35  ; 工位1-1 进托盘
      AND     X0A  ; 工位1-1 装载台内托盘检测
      AND     M0  ; 自动运行
      MPS
      ANI     M21
      SET     M20  ; 夹紧气缸推动
      MPP
      OUT     T40 D1022  ; 工位1-1托盘到位 / 工位到位延时
55    LD      M20  ; 夹紧气缸推动
      AND     X60  ; 工位1-1夹紧到位
      SET     M21
      RST     M20  ; 夹紧气缸推动
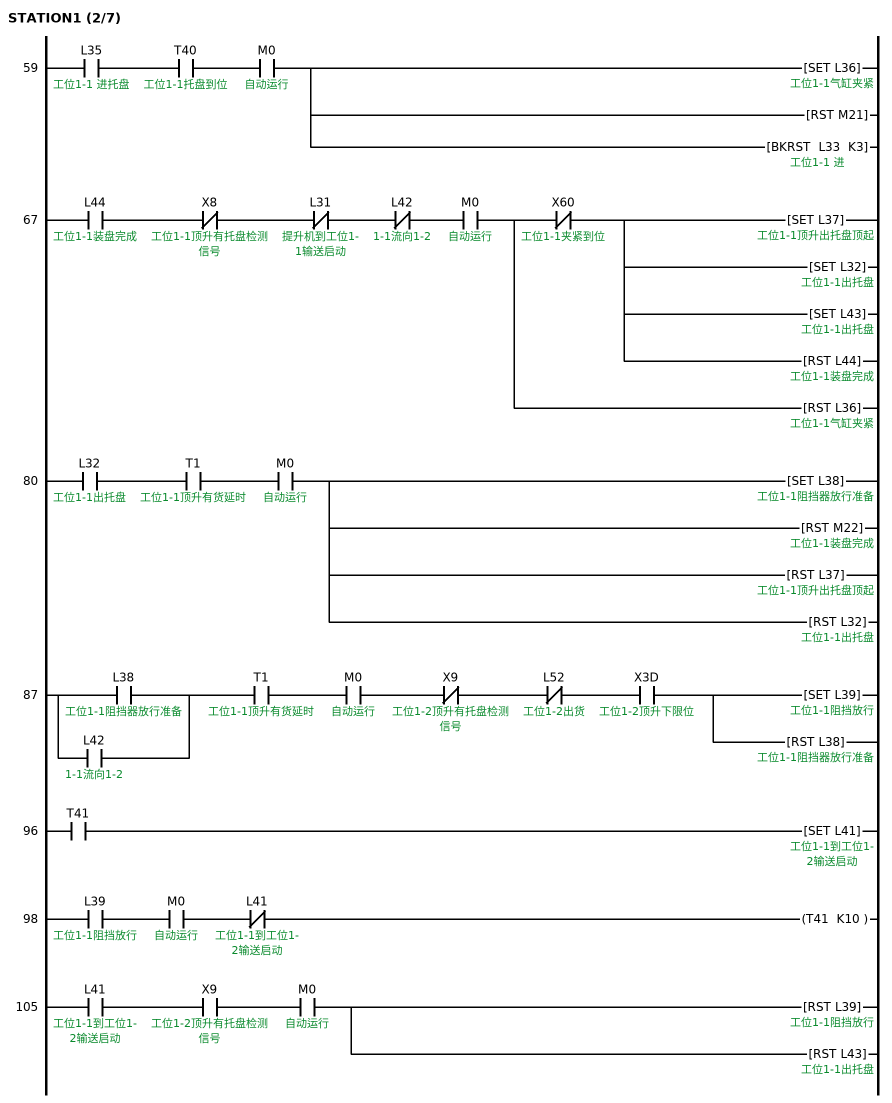
59    LD      L35  ; 工位1-1 进托盘
      AND     T40  ; 工位1-1托盘到位
      AND     M0  ; 自动运行
      SET     L36  ; 工位1-1气缸夹紧
      RST     M21
      BKRST   L33 K3
67    LD      L44  ; 工位1-1装盘完成
      ANI     X8  ; 工位1-1顶升有托盘检测信号
      ANI     L31  ; 提升机到工位1-1输送启动
      ANI     L42  ; 1-1流向1-2
      AND     M0  ; 自动运行
      MPS
      ANI     X60  ; 工位1-1夹紧到位
      SET     L37  ; 工位1-1顶升出托盘顶起
      SET     L32  ; 工位1-1出托盘
      SET     L43  ; 工位1-1出托盘
      RST     L44  ; 工位1-1装盘完成
      MPP
      RST     L36  ; 工位1-1气缸夹紧
80    LD      L32  ; 工位1-1出托盘
      AND     T1  ; 工位1-1顶升有货延时
      AND     M0  ; 自动运行
      SET     L38  ; 工位1-1阻挡器放行准备
      RST     M22  ; 工位1-1装盘完成
      RST     L37  ; 工位1-1顶升出托盘顶起
      RST     L32  ; 工位1-1出托盘
87    LD      L38  ; 工位1-1阻挡器放行准备
      OR      L42  ; 1-1流向1-2
      AND     T1  ; 工位1-1顶升有货延时
      AND     M0  ; 自动运行
      ANI     X9  ; 工位1-2顶升有托盘检测信号
      ANI     L52  ; 工位1-2出货
      AND     X3D  ; 工位1-2顶升下限位
      SET     L39  ; 工位1-1阻挡放行
      RST     L38  ; 工位1-1阻挡器放行准备
96    LD      T41
      SET     L41  ; 工位1-1到工位1-2输送启动
98    LD      L39  ; 工位1-1阻挡放行
      AND     M0  ; 自动运行
      ANI     L41  ; 工位1-1到工位1-2输送启动
      OUT     T41 K10
105   LD      L41  ; 工位1-1到工位1-2输送启动
      AND     X9  ; 工位1-2顶升有托盘检测信号
      AND     M0  ; 自动运行
      RST     L39  ; 工位1-1阻挡放行
      RST     L43  ; 工位1-1出托盘
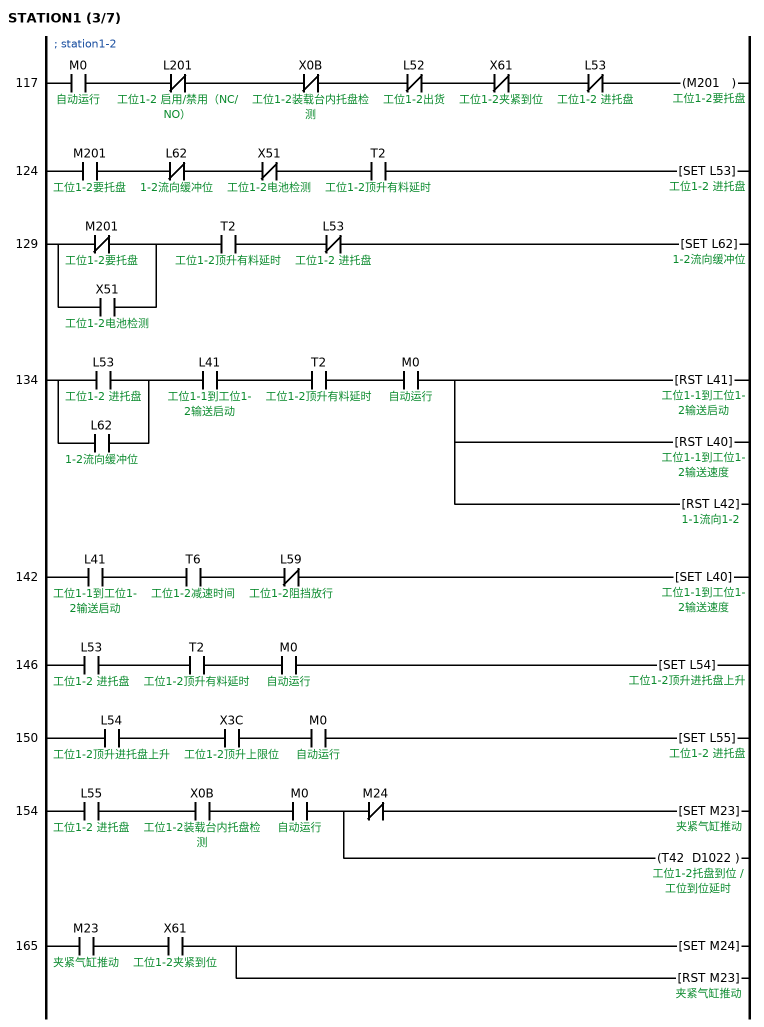
; station1-2
117   LD      M0  ; 自动运行
      ANI     L201  ; 工位1-2 启用/禁用（NC/NO）
      ANI     X0B  ; 工位1-2装载台内托盘检测
      ANI     L52  ; 工位1-2出货
      ANI     X61  ; 工位1-2夹紧到位
      ANI     L53  ; 工位1-2 进托盘
      OUT     M201  ; 工位1-2要托盘
124   LD      M201  ; 工位1-2要托盘
      ANI     L62  ; 1-2流向缓冲位
      ANI     X51  ; 工位1-2电池检测
      AND     T2  ; 工位1-2顶升有料延时
      SET     L53  ; 工位1-2 进托盘
129   LDI     M201  ; 工位1-2要托盘
      OR      X51  ; 工位1-2电池检测
      AND     T2  ; 工位1-2顶升有料延时
      ANI     L53  ; 工位1-2 进托盘
      SET     L62  ; 1-2流向缓冲位
134   LD      L53  ; 工位1-2 进托盘
      OR      L62  ; 1-2流向缓冲位
      AND     L41  ; 工位1-1到工位1-2输送启动
      AND     T2  ; 工位1-2顶升有料延时
      AND     M0  ; 自动运行
      RST     L41  ; 工位1-1到工位1-2输送启动
      RST     L40  ; 工位1-1到工位1-2输送速度
      RST     L42  ; 1-1流向1-2
142   LD      L41  ; 工位1-1到工位1-2输送启动
      AND     T6  ; 工位1-2减速时间
      ANI     L59  ; 工位1-2阻挡放行
      SET     L40  ; 工位1-1到工位1-2输送速度
146   LD      L53  ; 工位1-2 进托盘
      AND     T2  ; 工位1-2顶升有料延时
      AND     M0  ; 自动运行
      SET     L54  ; 工位1-2顶升进托盘上升
150   LD      L54  ; 工位1-2顶升进托盘上升
      AND     X3C  ; 工位1-2顶升上限位
      AND     M0  ; 自动运行
      SET     L55  ; 工位1-2 进托盘
154   LD      L55  ; 工位1-2 进托盘
      AND     X0B  ; 工位1-2装载台内托盘检测
      AND     M0  ; 自动运行
      MPS
      ANI     M24
      SET     M23  ; 夹紧气缸推动
      MPP
      OUT     T42 D1022  ; 工位1-2托盘到位 / 工位到位延时
165   LD      M23  ; 夹紧气缸推动
      AND     X61  ; 工位1-2夹紧到位
      SET     M24
      RST     M23  ; 夹紧气缸推动
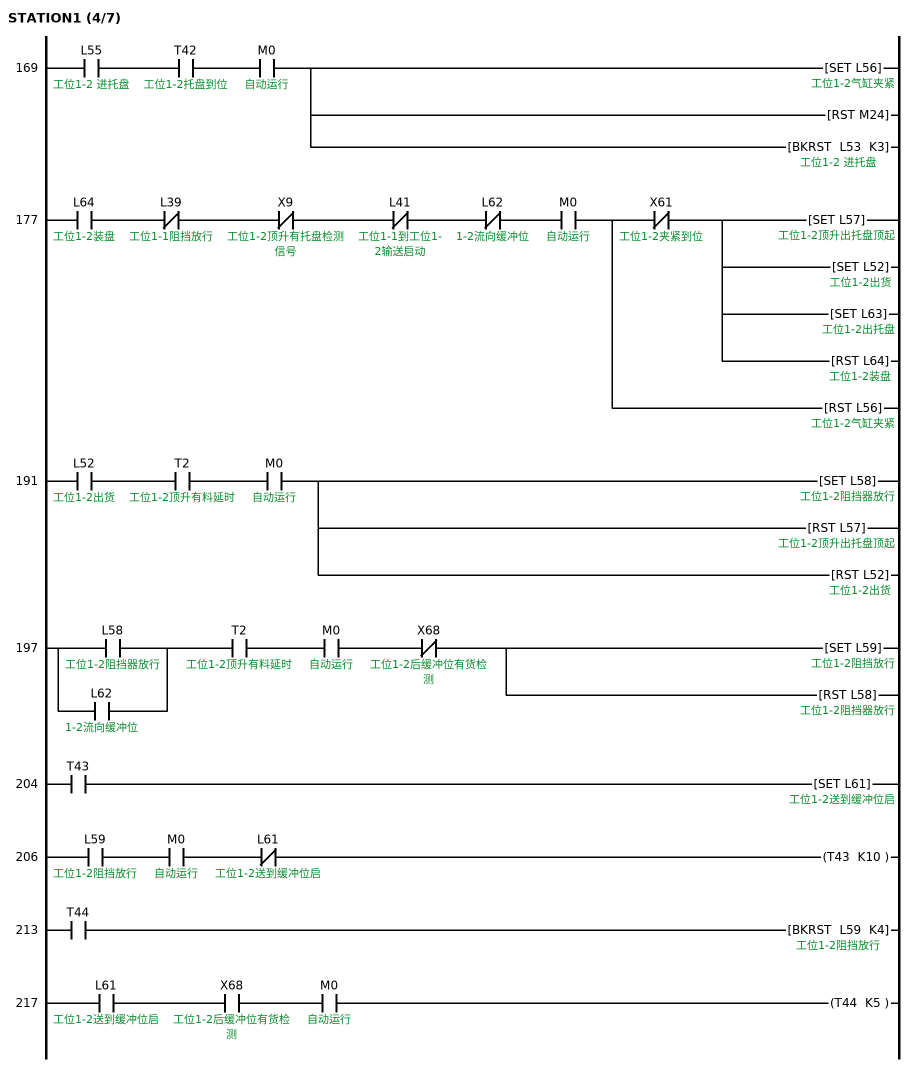
169   LD      L55  ; 工位1-2 进托盘
      AND     T42  ; 工位1-2托盘到位
      AND     M0  ; 自动运行
      SET     L56  ; 工位1-2气缸夹紧
      RST     M24
      BKRST   L53 K3
177   LD      L64  ; 工位1-2装盘
      ANI     L39  ; 工位1-1阻挡放行
      ANI     X9  ; 工位1-2顶升有托盘检测信号
      ANI     L41  ; 工位1-1到工位1-2输送启动
      ANI     L62  ; 1-2流向缓冲位
      AND     M0  ; 自动运行
      MPS
      ANI     X61  ; 工位1-2夹紧到位
      SET     L57  ; 工位1-2顶升出托盘顶起
      SET     L52  ; 工位1-2出货
      SET     L63  ; 工位1-2出托盘
      RST     L64  ; 工位1-2装盘
      MPP
      RST     L56  ; 工位1-2气缸夹紧
191   LD      L52  ; 工位1-2出货
      AND     T2  ; 工位1-2顶升有料延时
      AND     M0  ; 自动运行
      SET     L58  ; 工位1-2阻挡器放行
      RST     L57  ; 工位1-2顶升出托盘顶起
      RST     L52  ; 工位1-2出货
197   LD      L58  ; 工位1-2阻挡器放行
      OR      L62  ; 1-2流向缓冲位
      AND     T2  ; 工位1-2顶升有料延时
      AND     M0  ; 自动运行
      ANI     X68  ; 工位1-2后缓冲位有货检测
      SET     L59  ; 工位1-2阻挡放行
      RST     L58  ; 工位1-2阻挡器放行
204   LD      T43
      SET     L61  ; 工位1-2送到缓冲位启
206   LD      L59  ; 工位1-2阻挡放行
      AND     M0  ; 自动运行
      ANI     L61  ; 工位1-2送到缓冲位启
      OUT     T43 K10
213   LD      T44
      BKRST   L59 K4
217   LD      L61  ; 工位1-2送到缓冲位启
      AND     X68  ; 工位1-2后缓冲位有货检测
      AND     M0  ; 自动运行
      OUT     T44 K5
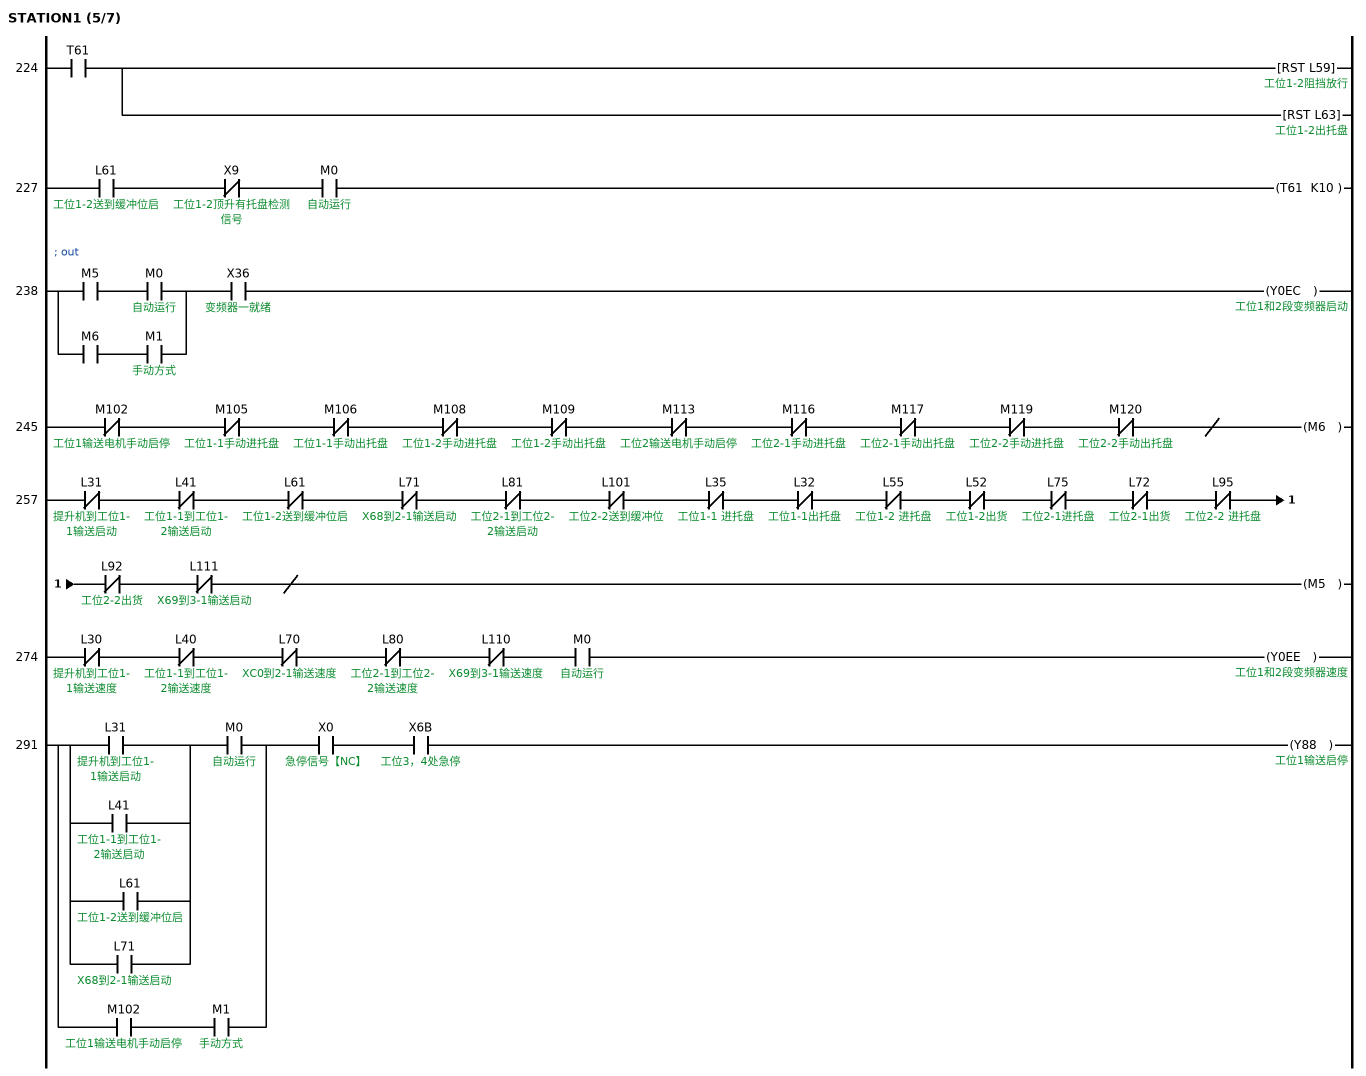
224   LD      T61
      RST     L59  ; 工位1-2阻挡放行
      RST     L63  ; 工位1-2出托盘
227   LD      L61  ; 工位1-2送到缓冲位启
      ANI     X9  ; 工位1-2顶升有托盘检测信号
      AND     M0  ; 自动运行
      OUT     T61 K10
; out
238   LD      M5
      AND     M0  ; 自动运行
      LD      M6
      AND     M1  ; 手动方式
      ORB
      AND     X36  ; 变频器一就绪
      OUT     Y0EC  ; 工位1和2段变频器启动
245   LDI     M102  ; 工位1输送电机手动启停
      ANI     M105  ; 工位1-1手动进托盘
      ANI     M106  ; 工位1-1手动出托盘
      ANI     M108  ; 工位1-2手动进托盘
      ANI     M109  ; 工位1-2手动出托盘
      ANI     M113  ; 工位2输送电机手动启停
      ANI     M116  ; 工位2-1手动进托盘
      ANI     M117  ; 工位2-1手动出托盘
      ANI     M119  ; 工位2-2手动进托盘
      ANI     M120  ; 工位2-2手动出托盘
      INV
      OUT     M6
257   LDI     L31  ; 提升机到工位1-1输送启动
      ANI     L41  ; 工位1-1到工位1-2输送启动
      ANI     L61  ; 工位1-2送到缓冲位启
      ANI     L71  ; X68到2-1输送启动
      ANI     L81  ; 工位2-1到工位2-2输送启动
      ANI     L101  ; 工位2-2送到缓冲位
      ANI     L35  ; 工位1-1 进托盘
      ANI     L32  ; 工位1-1出托盘
      ANI     L55  ; 工位1-2 进托盘
      ANI     L52  ; 工位1-2出货
      ANI     L75  ; 工位2-1进托盘
      ANI     L72  ; 工位2-1出货
      ANI     L95  ; 工位2-2 进托盘
      ANI     L92  ; 工位2-2出货
      ANI     L111  ; X69到3-1输送启动
      INV
      OUT     M5
274   LDI     L30  ; 提升机到工位1-1输送速度
      ANI     L40  ; 工位1-1到工位1-2输送速度
      ANI     L70  ; XC0到2-1输送速度
      ANI     L80  ; 工位2-1到工位2-2输送速度
      ANI     L110  ; X69到3-1输送速度
      AND     M0  ; 自动运行
      OUT     Y0EE  ; 工位1和2段变频器速度
        [note] ON高速，OFF低速
291   LD      L31  ; 提升机到工位1-1输送启动
      OR      L41  ; 工位1-1到工位1-2输送启动
      OR      L61  ; 工位1-2送到缓冲位启
      OR      L71  ; X68到2-1输送启动
      AND     M0  ; 自动运行
      LD      M102  ; 工位1输送电机手动启停
      AND     M1  ; 手动方式
      ORB
      AND     X0  ; 急停信号【NC】
      AND     X6B  ; 工位3，4处急停
      OUT     Y88  ; 工位1输送启停
        [note] 1-1
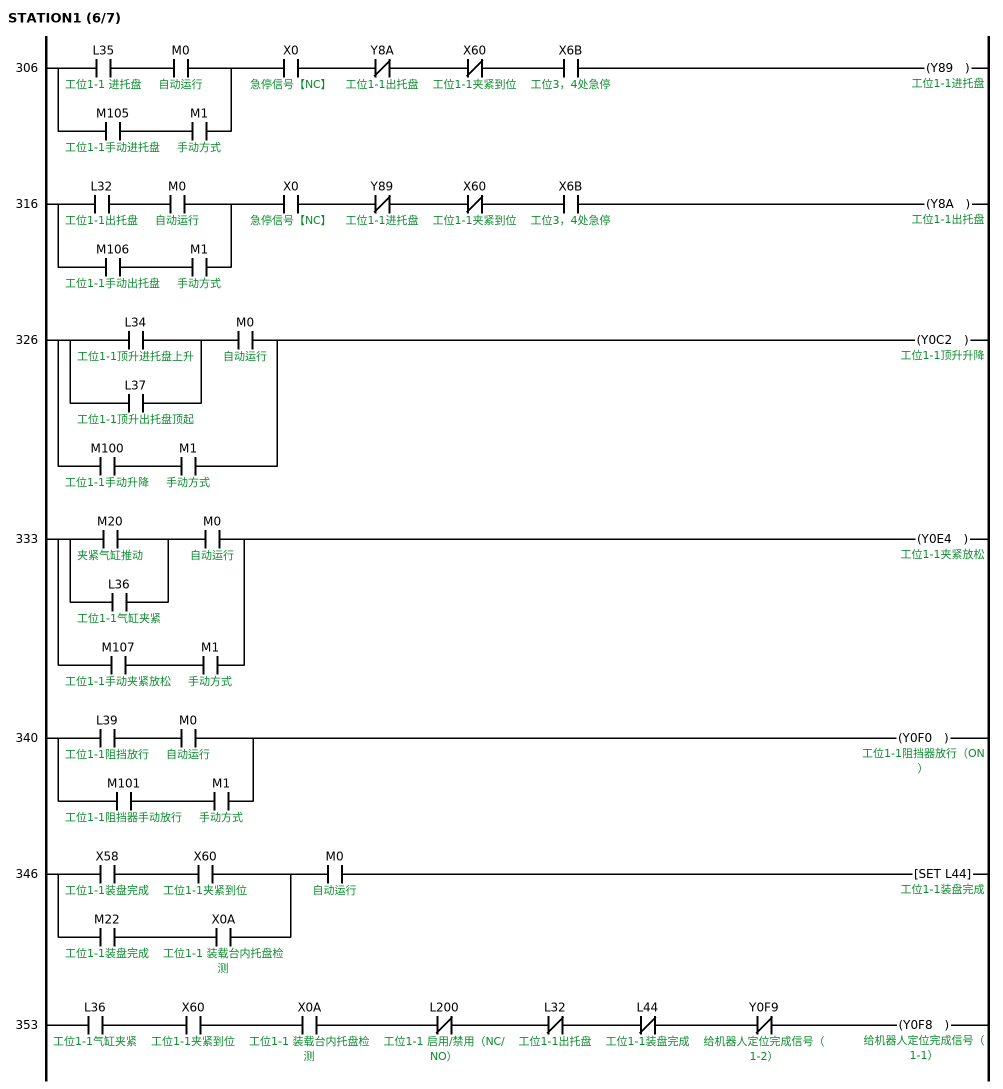
306   LD      L35  ; 工位1-1 进托盘
      AND     M0  ; 自动运行
      LD      M105  ; 工位1-1手动进托盘
      AND     M1  ; 手动方式
      ORB
      AND     X0  ; 急停信号【NC】
      ANI     Y8A  ; 工位1-1出托盘
      ANI     X60  ; 工位1-1夹紧到位
      AND     X6B  ; 工位3，4处急停
      OUT     Y89  ; 工位1-1进托盘
316   LD      L32  ; 工位1-1出托盘
      AND     M0  ; 自动运行
      LD      M106  ; 工位1-1手动出托盘
      AND     M1  ; 手动方式
      ORB
      AND     X0  ; 急停信号【NC】
      ANI     Y89  ; 工位1-1进托盘
      ANI     X60  ; 工位1-1夹紧到位
      AND     X6B  ; 工位3，4处急停
      OUT     Y8A  ; 工位1-1出托盘
326   LD      L34  ; 工位1-1顶升进托盘上升
      OR      L37  ; 工位1-1顶升出托盘顶起
      AND     M0  ; 自动运行
      LD      M100  ; 工位1-1手动升降
      AND     M1  ; 手动方式
      ORB
      OUT     Y0C2  ; 工位1-1顶升升降
333   LD      M20  ; 夹紧气缸推动
      OR      L36  ; 工位1-1气缸夹紧
      AND     M0  ; 自动运行
      LD      M107  ; 工位1-1手动夹紧放松
      AND     M1  ; 手动方式
      ORB
      OUT     Y0E4  ; 工位1-1夹紧放松
340   LD      L39  ; 工位1-1阻挡放行
      AND     M0  ; 自动运行
      LD      M101  ; 工位1-1阻挡器手动放行
      AND     M1  ; 手动方式
      ORB
      OUT     Y0F0  ; 工位1-1阻挡器放行（ON）
346   LD      X58  ; 工位1-1装盘完成
      AND     X60  ; 工位1-1夹紧到位
      LD      M22  ; 工位1-1装盘完成
      AND     X0A  ; 工位1-1 装载台内托盘检测
      ORB
      AND     M0  ; 自动运行
      SET     L44  ; 工位1-1装盘完成
353   LD      L36  ; 工位1-1气缸夹紧
      AND     X60  ; 工位1-1夹紧到位
      AND     X0A  ; 工位1-1 装载台内托盘检测
      ANI     L200  ; 工位1-1 启用/禁用（NC/NO）
      ANI     L32  ; 工位1-1出托盘
      ANI     L44  ; 工位1-1装盘完成
      ANI     Y0F9  ; 给机器人定位完成信号（1-2）
      OUT     Y0F8  ; 给机器人定位完成信号（1-1）
